// TIA Portal project "AC200_1.1" (V15.1)

(* hardware
DEVICE "S7-1200 station_1"  S7-1200 Station
   slot 0: "Rack_0"  S7-1200 Rack  Rack  V1.0
   slot 1: "PLC_1"  CPU 1215C DC/DC/Rly  6ES7 215-1HG40-0XB0  V4.2
   slot 2: "DI 8x24VDC/DQ 8xRelay_1"  SM 1223 DI8/DQ8 x relay  6ES7 223-1PH32-0XB0  V2.0
   slot 3: "DI 8x24VDC/DQ 8xRelay_2"  SM 1223 DI8/DQ8 x relay  6ES7 223-1PH32-0XB0  V2.0
   slot 4: "AI 4x16BIT_1"  SM 1231 AI4 x HF  6ES7 231-5ND32-0XB0  V2.0
   slot 101: "CM 1241 (RS232)_1"  6ES7 241-1AH32-0XB0  V2.2
DEVICE "HMI_1"  KTP700 Basic PN
   slot 0: "HMI_1"  KTP700 Basic PN  6AV2 123-2GB03-0AX0  15.1.0.0
   slot 1: "HMI_RT_1"  KTP700 Basic PN  6AV2 123-2GB03-0AX0  15.1.0.0
   slot 5: "HMI_1.IE_CP_1"  PROFINET Interface  15.0.1.0
      slot 1: "PROFINET Interface_1"  PROFINET Interface
         slot 1: "Port_1"  Port
*)

// ===== PLC "PLC_1"  CPU 1215C DC/DC/Rly =====

VAR_GLOBAL   // PLC tag table "DI_CPU"
   "DI_EStop_Chain_OK" AT %I0.0 : Bool;   // Nút dừng khẩn NC mắc nối tiếp
   "DI_Phase_OK" AT %I0.1 : Bool;   // Relay bảo vệ mất pha; 1 = nguồn 3 pha tốt
   "DI_Door1_Closed" AT %I0.2 : Bool;   // Công tắc hành trình cửa 1; 1 = cửa đóng
   "DI_Door2_Closed" AT %I0.3 : Bool;   // Công tắc hành trình cửa 2; 1 = cửa đóng
   "DI_Tank_Level_OK" AT %I0.4 : Bool;   // Cảm biến mức bồn nước cấp; 1 = đủ nước
   "DI_SG_Level_High" AT %I0.5 : Bool;   // Mức nước bình sinh hơi; 1 = đầy, 0 = mức thấp
   "DI_GasketPress_High" AT %I0.6 : Bool;   // Tiếp điểm thường mở áp suất cao gioăng cửa; 1 = đạt mức cao
   "DI_JacketPress_High" AT %I0.7 : Bool;   // Tiếp điểm thường mở áp suất cao jacket; 1 = đạt mức cao
   "DI_SGPress_High" AT %I1.0 : Bool;   // Tiếp điểm thường mở áp suất cao bình sinh hơi; 1 = đạt mức cao
   "DI_GasketPress_Low" AT %I1.1 : Bool;
END_VAR

VAR_GLOBAL   // PLC tag table "DI_SM1223_1"
   "DI_Door1_Open_PB" AT %I8.0 : Bool;   // Nút vật lý mở cửa 1
   "DI_Door1_Close_PB" AT %I8.1 : Bool;   // Nút vật lý đóng cửa 1
   "DI_Door2_Open_PB" AT %I8.2 : Bool;   // Nút vật lý mở cửa 2
   "DI_Door2_Close_PB" AT %I8.3 : Bool;   // Nút vật lý đóng cửa 2
   "DI_WaterPump_OL_OK" AT %I8.4 : Bool;   // Tiếp điểm NC relay nhiệt bơm nước; 1 = bình thường
   "DI_VacuumPump_OL_OK" AT %I8.5 : Bool;   // Tiếp điểm NC relay nhiệt bơm chân không; 1 = bình thường
END_VAR

VAR_GLOBAL   // PLC tag table "DO_CPU"
   "DO_Heater1" AT %Q0.0 : Bool;   // Điều khiển SSR cụm nhiệt 9 kW số 1
   "DO_Heater2" AT %Q0.1 : Bool;   // Điều khiển SSR cụm nhiệt 9 kW số 2
   "DO_Heater3" AT %Q0.2 : Bool;   // Điều khiển SSR cụm nhiệt 9 kW số 3
   "DO_WaterPump" AT %Q0.3 : Bool;   // Điều khiển contactor/relay bơm nước
   "DO_VacuumPump" AT %Q0.4 : Bool;   // Điều khiển contactor bơm chân không
   "DO_Door1_Open" AT %Q0.5 : Bool;   // Cuộn mở van 5/2 cửa 1
   "DO_Door1_Close" AT %Q0.6 : Bool;   // Cuộn đóng van 5/2 cửa 1
   "DO_Door2_Open" AT %Q0.7 : Bool;   // Cuộn mở van 5/2 cửa 2
   "DO_Door2_Close" AT %Q1.0 : Bool;   // Cuộn đóng van 5/2 cửa 2
   "DO_Buzzer" AT %Q1.1 : Bool;   // Còi báo 24 VDC
END_VAR

VAR_GLOBAL   // PLC tag table "DO_SM1223_2"
   "DO_WaterInlet_01" AT %Q12.0 : Bool;   // Van điện từ cấp nước NC số 1
   "DO_WaterDrain" AT %Q12.1 : Bool;   // Van điện từ xả nước/khí NO
   "DO_LampRun" AT %Q12.2 : Bool;   // Đèn Run - máy đang vận hành
   "DO_LampError" AT %Q12.3 : Bool;   // Đèn Error - hệ thống có lỗi
   "DO_LampDoor1" AT %Q12.4 : Bool;   // Đèn báo cửa 1 đã đóng an toàn
   "DO_LampDoor2" AT %Q12.5 : Bool;   // Đèn báo cửa 2 đã đóng an toàn
   "DO_WaterInlet_02" AT %Q12.6 : Bool;   // Van điện từ cấp nước NC số 2
END_VAR

VAR_GLOBAL   // PLC tag table "AI_SM1231"
   "AI_ChamberPressure1_Raw" AT %IW128 : Int;   // Áp suất buồng hấp vt1, 4-20 mA, -1...5 bar
   "AI_ChamberPressure2_Raw" AT %IW130 : Int;   // Áp suất buồng hấp vt2, 4-20 mA, -1...5 bar
   "AI_Temperature_Raw" AT %IW132 : Int;   // PT100 qua bộ chuyển đổi 0-10 V
END_VAR

VAR_GLOBAL   // PLC tag table "HMI_Command"
   "HMI_Cmd_Start" AT %M100.0 : Bool;   // Nút Start trên HMI
   "HMI_Cmd_Stop" AT %M100.1 : Bool;   // Dừng bình thường từ HMI
   "HMI_Cmd_Abort" AT %M100.2 : Bool;   // Hủy chu trình từ HMI
   "HMI_Cmd_AckAlarm" AT %M100.3 : Bool;   // Xác nhận cảnh báo và tắt còi
   "HMI_Cmd_Reset" AT %M100.4 : Bool;   // Reset lỗi khi điều kiện đã an toàn
   "HMI_Mode_Auto" AT %M100.5 : Bool;   // Yêu cầu chọn chế độ Auto
   "HMI_Mode_Manual" AT %M100.6 : Bool;   // Yêu cầu chọn chế độ Manual
   "HMI_Mode_Service" AT %M100.7 : Bool;   // Yêu cầu chọn chế độ Service; cần phân quyền
   "HMI_Cmd_Door1Open" AT %M101.0 : Bool;   // Yêu cầu mở cửa 1; PLC phải kiểm tra áp suất và liên động
   "HMI_Cmd_Door1Close" AT %M101.1 : Bool;   // Yêu cầu đóng cửa 1
   "HMI_Cmd_Door2Open" AT %M101.2 : Bool;   // Yêu cầu mở cửa 2; PLC phải kiểm tra áp suất và liên động
   "HMI_Cmd_Door2Close" AT %M101.3 : Bool;   // Yêu cầu đóng cửa 2
   "HMI_Cmd_Print" AT %M101.4 : Bool;   // Yêu cầu in kết quả chu trình
   "HMI_Cmd_ClearAlarmHistory" AT %M101.5 : Bool;   // Yêu cầu xóa lịch sử cảnh báo; cần phân quyền
   "HMI_Cmd_Login" AT %M101.6 : Bool;   // Yêu cầu đăng nhập
   "HMI_Cmd_Logout" AT %M101.7 : Bool;   // Yêu cầu đăng xuất
   "HMI_Cmd_EndAccepted" AT %M121.1 : Bool;
END_VAR

VAR_GLOBAL   // PLC tag table "HMI_Setpoint"
   "HMI_ProgramNumber" AT %MW102 : Int;   // Số chương trình P1-P6
   "HMI_PreVacCycles_SP" AT %MW104 : Int;   // Số lần tiền chân không
   "HMI_SterilizeTime_Min" AT %MW106 : Int;   // Thời gian tiệt trùng, phút
   "HMI_DryTime_Min" AT %MW108 : Int;   // Thời gian sấy, phút
   "HMI_Temperature_SP" AT %MD112 : Real;   // Nhiệt độ đặt, °C
   "HMI_Pressure_SP" AT %MD116 : Real;   // Áp suất đặt, bar
   "HMI_User_Str_Min" AT %MW110 : Int;
   "HMI_User_Dry_Min" AT %MW112 : Int;
   "HMI_User_Temp" AT %MW114 : Int;
END_VAR

VAR_GLOBAL   // PLC tag table "HMI_Status"
   "HMI_Sts_SystemReady" AT %M120.0 : Bool;   // Hệ thống sẵn sàng
   "HMI_Sts_CycleRunning" AT %M120.1 : Bool;   // Chu trình đang chạy
   "HMI_Sts_CycleComplete" AT %M120.2 : Bool;   // Chu trình hoàn thành
   "HMI_Sts_AlarmActive" AT %M120.3 : Bool;   // Đang có cảnh báo
   "HMI_Sts_Door1Closed" AT %M120.4 : Bool;   // Trạng thái cửa 1 đóng
   "HMI_Sts_Door2Closed" AT %M120.5 : Bool;   // Trạng thái cửa 2 đóng
   "HMI_Sts_HeaterRunning" AT %M120.6 : Bool;   // Gia nhiệt đang hoạt động
   "HMI_Sts_VacuumRunning" AT %M120.7 : Bool;   // Bơm chân không đang chạy
   "HMI_ProcessStep" AT %MW122 : Int;   // Mã bước quy trình hiện tại
   "HMI_Temperature_PV" AT %MD124 : Real;   // Nhiệt độ thực tế đã scale, °C
   "HMI_ChamberPressure_01_PV" AT %MD128 : Real;   // Áp suất thực tế buồng hấp tại vị trí 1 đã scale, bar
   "HMI_ChamberPressure_02_PV" AT %MD132 : Real;   // Áp suất thực tế buồng hấp tại vị trí 2 đã scale, bar
   "HMI_RemainingTime_Sec" AT %MD136 : DInt;   // Thời gian còn lại, giây
   "HMI_AlarmErrorWord" AT %MW168 : Int;   // mã loi
   "HMI_ChamberPressure_com" AT %MD144 : Real;   // Ap sau trung binh
   "HMI_Sts_Dry_Enable" AT %M121.0 : Bool;
   "HMI_AlarmWarningWord" AT %MW170 : Int;   // ma canh bao
   "HMI_AlarmAckWord" AT %MW172 : Int;
   "HMI_Sts_BuzzerRequest" AT %M174.0 : Bool;
   "HMI_Sts_LampErrorRequest" AT %M174.1 : Bool;
   "HMI_StartBlockReason" AT %MW174 : Int;
   "HMI_StartBlocked" AT %M174.2 : Bool;
   "HMI_PageRequest" AT %MW176 : Int;
   "HMI_SelectedProgram" AT %MW178 : Int;
END_VAR

VAR_GLOBAL   // PLC tag table "HMI_Manual"
   "HMI_Man_WaterPump" AT %M150.0 : Bool;   // Yêu cầu chạy tay bơm nước; chỉ có hiệu lực trong Service và đủ liên động
   "HMI_Man_VacuumPump" AT %M150.1 : Bool;   // Yêu cầu chạy tay bơm chân không
   "HMI_Man_Heater1" AT %M150.2 : Bool;   // Yêu cầu gia nhiệt tay cụm 1; phải có nước và điều kiện an toàn
   "HMI_Man_Heater2" AT %M150.3 : Bool;   // Yêu cầu gia nhiệt tay cụm 2; phải có nước và điều kiện an toàn
   "HMI_Man_Heater3" AT %M150.4 : Bool;   // Yêu cầu gia nhiệt tay cụm 3; phải có nước và điều kiện an toàn
   "HMI_Man_PilotValve_01" AT %M151.0 : Bool;   // Yêu cầu điều khiển tay van pilot V1; PLC vẫn kiểm tra liên động
   "HMI_Man_PilotValve_02" AT %M151.1 : Bool;   // Yêu cầu điều khiển tay van pilot V2; PLC vẫn kiểm tra liên động
   "HMI_Man_PilotValve_03" AT %M151.2 : Bool;   // Yêu cầu điều khiển tay van pilot V3; PLC vẫn kiểm tra liên động
   "HMI_Man_PilotValve_04" AT %M151.3 : Bool;   // Yêu cầu điều khiển tay van pilot V4; PLC vẫn kiểm tra liên động
   "HMI_Man_PilotValve_05" AT %M151.4 : Bool;   // Yêu cầu điều khiển tay van pilot V5; PLC vẫn kiểm tra liên động
   "HMI_Man_PilotValve_06" AT %M151.5 : Bool;   // Yêu cầu điều khiển tay van pilot V6; PLC vẫn kiểm tra liên động
   "HMI_Man_PilotValve_07" AT %M151.6 : Bool;   // Yêu cầu điều khiển tay van pilot V7; PLC vẫn kiểm tra liên động
   "HMI_Man_PilotValve_08" AT %M151.7 : Bool;   // Yêu cầu điều khiển tay van pilot V8; PLC vẫn kiểm tra liên động
   "HMI_Man_WaterInlet_01" AT %M152.0 : Bool;   // Yêu cầu điều khiển tay van cấp nước 1
   "HMI_Man_WaterDrain" AT %M152.1 : Bool;   // Yêu cầu điều khiển tay van xả
   "HMI_Man_BuzzerTest" AT %M152.2 : Bool;   // Nút thử còi
   "HMI_Man_WaterInlet_02" AT %M152.3 : Bool;   // Yêu cầu chạy thử van cấp nước số 2
END_VAR

VAR_GLOBAL   // PLC tag table "DO_SM1223_1"
   "DO_PilotValve_01" AT %Q8.0 : Bool;   // Van pilot điều khiển van xiên V1
   "DO_PilotValve_02" AT %Q8.1 : Bool;   // Van pilot điều khiển van xiên V2
   "DO_PilotValve_03" AT %Q8.2 : Bool;   // Van pilot điều khiển van xiên V3
   "DO_PilotValve_04" AT %Q8.3 : Bool;   // Van pilot điều khiển van xiên V4/NO
   "DO_PilotValve_05" AT %Q8.4 : Bool;   // Van pilot điều khiển van xiên V5/NO
   "DO_PilotValve_06" AT %Q8.5 : Bool;   // Van pilot điều khiển van xiên V6/NO
   "DO_PilotValve_07" AT %Q8.6 : Bool;   // Van pilot điều khiển van xiên V7/NO
   "DO_PilotValve_08" AT %Q8.7 : Bool;   // Van pilot điều khiển van xiên V8
END_VAR

VAR_GLOBAL   // PLC tag table "Auto_Output"
   "AUTO_Q_Heater1" AT %M164.0 : Bool;   // Đầu ra trung gian Auto cho heater 1; không ghi trực tiếp %Q
   "AUTO_Q_Heater2" AT %M164.1 : Bool;   // Đầu ra trung gian Auto cho heater 2; không ghi trực tiếp %Q
   "AUTO_Q_Heater3" AT %M164.2 : Bool;   // Đầu ra trung gian Auto cho heater 3; không ghi trực tiếp %Q
   "AUTO_Q_WaterPump" AT %M164.3 : Bool;   // Đầu ra trung gian Auto cho bơm nước
   "AUTO_Q_VacuumPump" AT %M164.4 : Bool;   // Đầu ra trung gian Auto cho bơm chân không
   "AUTO_Q_PilotValve_01" AT %M164.5 : Bool;   // Đầu ra trung gian Auto cho van pilot 01
   "AUTO_Q_PilotValve_02" AT %M164.6 : Bool;   // Đầu ra trung gian Auto cho van pilot 02
   "AUTO_Q_PilotValve_03" AT %M164.7 : Bool;   // Đầu ra trung gian Auto cho van pilot 03
   "AUTO_Q_PilotValve_04" AT %M165.0 : Bool;   // Đầu ra trung gian Auto cho van pilot 04
   "AUTO_Q_PilotValve_05" AT %M165.1 : Bool;   // Đầu ra trung gian Auto cho van pilot 05
   "AUTO_Q_PilotValve_06" AT %M165.2 : Bool;   // Đầu ra trung gian Auto cho van pilot 06
   "AUTO_Q_PilotValve_07" AT %M165.3 : Bool;   // Đầu ra trung gian Auto cho van pilot 07
   "AUTO_Q_PilotValve_08" AT %M165.4 : Bool;   // Đầu ra trung gian Auto cho van pilot 08
   "AUTO_Q_WaterInlet_01" AT %M165.5 : Bool;   // Đầu ra trung gian Auto cho van cấp nước 01
   "AUTO_Q_WaterInlet_02" AT %M165.6 : Bool;   // Đầu ra trung gian Auto cho van cấp nước 02
   "AUTO_Q_WaterDrain" AT %M165.7 : Bool;   // Đầu ra trung gian Auto cho van xả nước/khí
   "AUTO_Q_Buzzer" AT %M166.0 : Bool;   // Đầu ra trung gian Auto cho còi báo
   "AUTO_Cmd_Start" AT %M166.1 : Bool;
END_VAR

VAR_GLOBAL   // PLC tag table "Manual_Output"
   "MAN_Q_Heater1" AT %M161.0 : Bool;   // Đầu ra trung gian Manual cho heater 1; không ghi trực tiếp %Q
   "MAN_Q_Heater2" AT %M161.1 : Bool;   // Đầu ra trung gian Manual cho heater 2; không ghi trực tiếp %Q
   "MAN_Q_Heater3" AT %M161.2 : Bool;   // Đầu ra trung gian Manual cho heater 3; không ghi trực tiếp %Q
   "MAN_Q_WaterPump" AT %M161.3 : Bool;   // Đầu ra trung gian Manual cho bơm nước
   "MAN_Q_VacuumPump" AT %M161.4 : Bool;   // Đầu ra trung gian Manual cho bơm chân không
   "MAN_Q_PilotValve_01" AT %M161.5 : Bool;   // Đầu ra trung gian Manual cho van pilot 01
   "MAN_Q_PilotValve_02" AT %M161.6 : Bool;   // Đầu ra trung gian Manual cho van pilot 02
   "MAN_Q_PilotValve_03" AT %M161.7 : Bool;   // Đầu ra trung gian Manual cho van pilot 03
   "MAN_Q_PilotValve_04" AT %M162.0 : Bool;   // Đầu ra trung gian Manual cho van pilot 04
   "MAN_Q_PilotValve_05" AT %M162.1 : Bool;   // Đầu ra trung gian Manual cho van pilot 05
   "MAN_Q_PilotValve_06" AT %M162.2 : Bool;   // Đầu ra trung gian Manual cho van pilot 06
   "MAN_Q_PilotValve_07" AT %M162.3 : Bool;   // Đầu ra trung gian Manual cho van pilot 07
   "MAN_Q_PilotValve_08" AT %M162.4 : Bool;   // Đầu ra trung gian Manual cho van pilot 08
   "MAN_Q_WaterInlet_01" AT %M162.5 : Bool;   // Đầu ra trung gian Manual cho van cấp nước 01
   "MAN_Q_WaterInlet_02" AT %M162.6 : Bool;   // Đầu ra trung gian Manual cho van cấp nước 02
   "MAN_Q_WaterDrain" AT %M162.7 : Bool;   // Đầu ra trung gian Manual cho van xả nước/khí
   "MAN_Q_Buzzer" AT %M163.0 : Bool;   // Đầu ra trung gian Manual cho thử còi
END_VAR

VAR_GLOBAL   // PLC tag table "SIG"
   "SIG_PressureMismatch" AT %M140.0 : Bool;
   "SIG_GasketTimeout" AT %M140.1 : Bool;
   "SIG_Vacuum Timeout" AT %M140.2 : Bool;
   "SIG_Heating Timeout" AT %M140.3 : Bool;
   "SIG_Sterilize TempLow" AT %M140.4 : Bool;
   "SIG_SGFillTimeout" AT %M140.5 : Bool;
   "SIG_ExhaustTimeout" AT %M140.6 : Bool;
   "SIG_Maintenance Due" AT %M140.7 : Bool;
   "SIG_HMICommunicationFault" AT %M141.0 : Bool;
   "SIG_PrinterFault" AT %M141.1 : Bool;
END_VAR

TYPE "UDT_AC200L_AutoConfig"
   STRUCT
      VacuumTarget_bar : Real := -0.75;
      VacuumFallback_bar : Real := -0.65;
      AllowVacuumFallback : Bool := TRUE;
      VacuumTimeout : Time := T#3M;
      ChargeTarget_bar : Real := 0.5;
      ChargeTimeout : Time := T#0MS;   // REQUIRED: not yet specified
      GasketTimeout : Time := T#3M;
      JacketTimeout : Time := T#3M;
      HeatTimeout : Time := T#35M;
      PIDApproach_C : Real := 10.0;
      JacketDrainTime : Time := T#4M;
      SterilizeStableTime : Time := T#0MS;   // REQUIRED
      SterilizePressureMin_bar : Real := 0.0;   // REQUIRED
      SterilizePressureMax_bar : Real := 0.0;   // REQUIRED
      TempLowOffset_C : Real := 1.2;
      TempLowTimeout : Time := T#3M;
      ExhaustTarget_bar : Real := 0.15;
      ExhaustTimeout : Time := T#5M;
      DryTarget_bar : Real := -0.65;
      DryAcquireTimeout : Time := T#0MS;   // REQUIRED
      BalanceTimeout : Time := T#0MS;   // REQUIRED
      ValveSettleTime : Time := T#0MS;   // REQUIRED: mechanical travel time
      PressureSafeBand_bar : Real := 0.15;
      PIDConfigured : Bool := FALSE;   // Set only after PID_Compact configuration
      RecoveryConfigured : Bool := FALSE;   // Confirm recovery exhaust routing
      RunPage : Int := 12;
      EndPage : Int := 15;   // Keep supplied DEMO value, verify actual HMI page
   END_STRUCT;
END_TYPE

DATA_BLOCK "FB_ManualTest_DB"   // DB1
{ S7_Optimized_Access := 'TRUE' }
VERSION : 0.4
// stored: InstanceOfName FB_ManualTest
"FB_ManualTest"
BEGIN
END_DATA_BLOCK

DATA_BLOCK "FB_AC200L_AlarmDirect_V7_DB"   // DB2
{ S7_Optimized_Access := 'TRUE' }
VERSION : 0.1
// stored: InstanceOfName FB_AC200L_AlarmDirect_V7
"FB_AC200L_AlarmDirect_V7"
BEGIN
END_DATA_BLOCK

DATA_BLOCK "FB_AnalogScale_DB"   // DB3
{ S7_Optimized_Access := 'TRUE' }
VERSION : 0.1
// stored: InstanceOfName FB_AnalogScale
"FB_AnalogScale"
BEGIN
END_DATA_BLOCK

DATA_BLOCK "FB_SGStartupFill_DB"   // DB4
{ S7_Optimized_Access := 'TRUE' }
VERSION : 0.5
// stored: InstanceOfName FB_SGStartupFill
"FB_SGStartupFill"
BEGIN
END_DATA_BLOCK

DATA_BLOCK "FB_StartPrecheck_DB"   // DB5
{ S7_Optimized_Access := 'TRUE' }
VERSION : 0.4
// stored: InstanceOfName FB_StartPrecheck
"FB_StartPrecheck"
BEGIN
END_DATA_BLOCK

DATA_BLOCK "FB_AutoCycle_Demo_DB"   // DB6
{ S7_Optimized_Access := 'TRUE' }
VERSION : 0.1
// stored: InstanceOfName FB_AutoCycle_Demo
"FB_AutoCycle_Demo"
BEGIN
END_DATA_BLOCK

DATA_BLOCK "FB_DoorControl_DB"   // DB7
{ S7_Optimized_Access := 'TRUE' }
VERSION : 1.2
// stored: InstanceOfName FB_DoorControl
"FB_DoorControl"
BEGIN
END_DATA_BLOCK

DATA_BLOCK "FB_AutoCycle_Main_DB"   // DB8
{ S7_Optimized_Access := 'TRUE' }
VERSION : 1.3
// stored: InstanceOfName FB_AutoCycle_Main
"FB_AutoCycle_Main"
BEGIN
END_DATA_BLOCK

DATA_BLOCK "DB_AC200L_AutoConfig"   // DB9
{ S7_Optimized_Access := 'TRUE' }
VERSION : 1.0
   VAR
      Settings : "UDT_AC200L_AutoConfig";
   END_VAR
BEGIN
END_DATA_BLOCK

FUNCTION_BLOCK "FB_ManualTest"   // FB1, SCL
{ S7_Optimized_Access := 'TRUE' }
VERSION : 0.4
   VAR_INPUT
      Enable : Bool;
      EStop_OK : Bool;
      Phase_OK : Bool;
      SG_Level_High : Bool;
      WaterPump_OL_OK : Bool;
      VacuumPump_OL_OK : Bool;
      Cmd_Heater1 : Bool;
      Cmd_Heater2 : Bool;
      Cmd_Heater3 : Bool;
      Cmd_WaterPump : Bool;
      Cmd_VacuumPump : Bool;
      Cmd_PilotValve_01 : Bool;
      Cmd_PilotValve_02 : Bool;
      Cmd_PilotValve_03 : Bool;
      Cmd_PilotValve_04 : Bool;
      Cmd_PilotValve_05 : Bool;
      Cmd_PilotValve_06 : Bool;
      Cmd_PilotValve_07 : Bool;
      Cmd_PilotValve_08 : Bool;
      Cmd_WaterInlet_01 : Bool;
      Cmd_WaterInlet_02 : Bool;
      Cmd_WaterDrain : Bool;
      Cmd_Buzzer : Bool;
   END_VAR
   VAR_OUTPUT
      Manual_Ready : Bool;
      Any_Command : Bool;
      Any_Output : Bool;
      Command_Blocked : Bool;
      MoreThanOneCommand : Bool;
      Safety_Trip : Bool;
      Q_Heater1 : Bool;
      Q_Heater2 : Bool;
      Q_Heater3 : Bool;
      Q_WaterPump : Bool;
      Q_VacuumPump : Bool;
      Q_PilotValve_01 : Bool;
      Q_PilotValve_02 : Bool;
      Q_PilotValve_03 : Bool;
      Q_PilotValve_04 : Bool;
      Q_PilotValve_05 : Bool;
      Q_PilotValve_06 : Bool;
      Q_PilotValve_07 : Bool;
      Q_PilotValve_08 : Bool;
      Q_WaterInlet_01 : Bool;
      Q_WaterInlet_02 : Bool;
      Q_WaterDrain : Bool;
      Q_Buzzer : Bool;
   END_VAR
   VAR_TEMP
      CommandCount : Int;
      TestPermit : Bool;
   END_VAR
BEGIN

   #CommandCount := 0;
   IF #Cmd_Heater1 THEN
       #CommandCount := #CommandCount + 1;
   END_IF;
   IF #Cmd_Heater2 THEN
       #CommandCount := #CommandCount + 1;
   END_IF;
   IF #Cmd_Heater3 THEN
       #CommandCount := #CommandCount + 1;
   END_IF;
   IF #Cmd_WaterPump THEN
       #CommandCount := #CommandCount + 1;
   END_IF;
   IF #Cmd_VacuumPump THEN
       #CommandCount := #CommandCount + 1;
   END_IF;
   IF #Cmd_PilotValve_01 THEN
       #CommandCount := #CommandCount + 1;
   END_IF;
   IF #Cmd_PilotValve_02 THEN
       #CommandCount := #CommandCount + 1;
   END_IF;
   IF #Cmd_PilotValve_03 THEN
       #CommandCount := #CommandCount + 1;
   END_IF;
   IF #Cmd_PilotValve_04 THEN
       #CommandCount := #CommandCount + 1;
   END_IF;
   IF #Cmd_PilotValve_05 THEN
       #CommandCount := #CommandCount + 1;
   END_IF;
   IF #Cmd_PilotValve_06 THEN
       #CommandCount := #CommandCount + 1;
   END_IF;
   IF #Cmd_PilotValve_07 THEN
       #CommandCount := #CommandCount + 1;
   END_IF;
   IF #Cmd_PilotValve_08 THEN
       #CommandCount := #CommandCount + 1;
   END_IF;
   IF #Cmd_WaterInlet_01 THEN
       #CommandCount := #CommandCount + 1;
   END_IF;
   IF #Cmd_WaterInlet_02 THEN
       #CommandCount := #CommandCount + 1;
   END_IF;
   IF #Cmd_WaterDrain THEN
       #CommandCount := #CommandCount + 1;
   END_IF;
   IF #Cmd_Buzzer THEN
       #CommandCount := #CommandCount + 1;
   END_IF;
   #Any_Command := #CommandCount > 0;
   #MoreThanOneCommand := #CommandCount > 1;
   #Manual_Ready := #Enable AND #EStop_OK AND #Phase_OK;
   #Safety_Trip := #Enable AND (NOT #EStop_OK OR NOT #Phase_OK);
   #TestPermit := #Manual_Ready;
   #Q_Heater1 := #TestPermit AND #Cmd_Heater1
   AND #SG_Level_High;
   #Q_Heater2 := #TestPermit AND #Cmd_Heater2
   AND #SG_Level_High;
   #Q_Heater3 := #TestPermit AND #Cmd_Heater3
   AND #SG_Level_High;
   #Q_WaterPump := #TestPermit AND #Cmd_WaterPump
   AND #WaterPump_OL_OK;
   #Q_VacuumPump := #TestPermit AND #Cmd_VacuumPump
   AND #VacuumPump_OL_OK;
   #Q_PilotValve_01 := #TestPermit AND #Cmd_PilotValve_01;
   #Q_PilotValve_02 := #TestPermit AND #Cmd_PilotValve_02;
   #Q_PilotValve_03 := #TestPermit AND #Cmd_PilotValve_03;
   #Q_PilotValve_04 := #TestPermit AND #Cmd_PilotValve_04;
   #Q_PilotValve_05 := #TestPermit AND #Cmd_PilotValve_05;
   #Q_PilotValve_06 := #TestPermit AND #Cmd_PilotValve_06;
   #Q_PilotValve_07 := #TestPermit AND #Cmd_PilotValve_07;
   #Q_PilotValve_08 := #TestPermit AND #Cmd_PilotValve_08;
   #Q_WaterInlet_01 := #TestPermit AND #Cmd_WaterInlet_01;
   #Q_WaterInlet_02 := #TestPermit AND #Cmd_WaterInlet_02;
   #Q_WaterDrain := #TestPermit AND #Cmd_WaterDrain;
   #Q_Buzzer := #TestPermit AND #Cmd_Buzzer;
   #Any_Output := #Q_Heater1 OR #Q_Heater2 OR #Q_Heater3
   OR #Q_WaterPump OR #Q_VacuumPump
   OR #Q_PilotValve_01 OR #Q_PilotValve_02
   OR #Q_PilotValve_03 OR #Q_PilotValve_04
   OR #Q_PilotValve_05 OR #Q_PilotValve_06
   OR #Q_PilotValve_07 OR #Q_PilotValve_08
   OR #Q_WaterInlet_01 OR #Q_WaterInlet_02
   OR #Q_WaterDrain OR #Q_Buzzer;
   #Command_Blocked := #Enable AND #Any_Command AND NOT #Any_Output;
END_FUNCTION_BLOCK

FUNCTION_BLOCK "FB_AC200L_AlarmDirect_V7"   // FB2, SCL
{ S7_Optimized_Access := 'TRUE' }
VERSION : 0.1
   VAR_INPUT
      DI_EStop_Chain_OK : Bool;
      DI_Phase_OK : Bool;
      DI_WaterPump_OL_OK : Bool;
      DI_VacuumPump_OL_OK : Bool;
      DI_Tank_Level_OK : Bool;
      DI_Door1_Closed : Bool;
      DI_Door2_Closed : Bool;
      DI_Door1_Open_PB : Bool;
      DI_Door2_Open_PB : Bool;
      AI_Temperature_Raw : Int;
      AI_ChamberPressure1_Raw : Int;
      AI_ChamberPressure2_Raw : Int;
      HMI_Temperature_PV : Real;
      HMI_ChamberPressure_01_PV : Real;
      HMI_ChamberPressure_02_PV : Real;
      HMI_Cmd_Start : Bool;
      HMI_Sts_CycleRunning : Bool;
      SIG_GasketTimeout : Bool;
      SIG_VacuumTimeout : Bool;
      SIG_HeatingTimeout : Bool;
      SIG_SterilizeTempLow : Bool;
      SIG_SGFillTimeout : Bool;
      SIG_ExhaustTimeout : Bool;
      SIG_MaintenanceDue : Bool;
      SIG_HMICommunicationFault : Bool;
      SIG_PrinterFault : Bool;
      SIG_PressureMismatch : Bool;
   END_VAR
   VAR_OUTPUT
      AlarmErrorWord : Int;
      AlarmWarningWord : Int;
      ErrorActive : Bool;
      WarningActive : Bool;
      AlarmActive : Bool;
      LampErrorRequest : Bool;
      BuzzerRequest : Bool;
   END_VAR
   VAR_IN_OUT
      AlarmAckWord : Int;
   END_VAR
   VAR
      TankLowTimer : TON_TIME;
   END_VAR
   VAR_TEMP
      UnackError : Bool;
   END_VAR
BEGIN
       #AlarmErrorWord.%X0 := NOT #DI_EStop_Chain_OK;
       #AlarmErrorWord.%X1 := NOT #DI_Phase_OK;
       #AlarmErrorWord.%X2 := NOT #DI_WaterPump_OL_OK;
       #AlarmErrorWord.%X3 := NOT #DI_VacuumPump_OL_OK;
       #AlarmErrorWord.%X4 := #HMI_Temperature_PV > 138.0;

       #TankLowTimer(
                     IN := NOT #DI_Tank_Level_OK,
                     PT := T#15s
       );

       #AlarmErrorWord.%X5 := #TankLowTimer.Q;

       #AlarmErrorWord.%X6 := (#AI_Temperature_Raw < 0)
       OR (#AI_Temperature_Raw > 27648);

       #AlarmErrorWord.%X7 := (#AI_ChamberPressure1_Raw < 0)
       OR (#AI_ChamberPressure1_Raw > 27648);

       #AlarmErrorWord.%X8 := (#AI_ChamberPressure2_Raw < 0)
       OR (#AI_ChamberPressure2_Raw > 27648);

       #AlarmErrorWord.%X9 := #SIG_PressureMismatch;
       #AlarmErrorWord.%X10 := #SIG_GasketTimeout;
       #AlarmErrorWord.%X11 := #SIG_VacuumTimeout;
       #AlarmErrorWord.%X12 := #SIG_HeatingTimeout;
       #AlarmErrorWord.%X13 := #SIG_SterilizeTempLow;
       #AlarmErrorWord.%X14 := #SIG_SGFillTimeout;
       #AlarmErrorWord.%X15 := #SIG_ExhaustTimeout;

       #AlarmWarningWord.%X0 := #HMI_Sts_CycleRunning
       AND #DI_Door1_Open_PB;

       #AlarmWarningWord.%X1 := #HMI_Sts_CycleRunning
       AND #DI_Door2_Open_PB;

       #AlarmWarningWord.%X2 := #HMI_Cmd_Start
       AND ((NOT #DI_Door1_Closed)
       OR (NOT #DI_Door2_Closed));

       #AlarmWarningWord.%X3 := (#DI_Door1_Open_PB OR #DI_Door2_Open_PB)
       AND ((#HMI_ChamberPressure_01_PV < -0.15)
       OR (#HMI_ChamberPressure_01_PV > 0.15)
       OR (#HMI_ChamberPressure_02_PV < -0.15)
       OR (#HMI_ChamberPressure_02_PV > 0.15));

       #AlarmWarningWord.%X4 := #SIG_MaintenanceDue;
       #AlarmWarningWord.%X5 := #SIG_HMICommunicationFault;
       #AlarmWarningWord.%X6 := #SIG_PrinterFault;
       #AlarmWarningWord.%X7 := FALSE;
       #AlarmWarningWord.%X8 := FALSE;
       #AlarmWarningWord.%X9 := FALSE;
       #AlarmWarningWord.%X10 := FALSE;
       #AlarmWarningWord.%X11 := FALSE;
       #AlarmWarningWord.%X12 := FALSE;
       #AlarmWarningWord.%X13 := FALSE;
       #AlarmWarningWord.%X14 := FALSE;
       #AlarmWarningWord.%X15 := FALSE;

       #ErrorActive := #AlarmErrorWord.%X0
       OR #AlarmErrorWord.%X1
       OR #AlarmErrorWord.%X2
       OR #AlarmErrorWord.%X3
       OR #AlarmErrorWord.%X4
       OR #AlarmErrorWord.%X5
       OR #AlarmErrorWord.%X6
       OR #AlarmErrorWord.%X7
       OR #AlarmErrorWord.%X8
       OR #AlarmErrorWord.%X9
       OR #AlarmErrorWord.%X10
       OR #AlarmErrorWord.%X11
       OR #AlarmErrorWord.%X12
       OR #AlarmErrorWord.%X13
       OR #AlarmErrorWord.%X14
       OR #AlarmErrorWord.%X15;

       #WarningActive := #AlarmWarningWord.%X0
       OR #AlarmWarningWord.%X1
       OR #AlarmWarningWord.%X2
       OR #AlarmWarningWord.%X3
       OR #AlarmWarningWord.%X4
       OR #AlarmWarningWord.%X5
       OR #AlarmWarningWord.%X6;

       #AlarmActive := #ErrorActive OR #WarningActive;

       #AlarmAckWord.%X0 := #AlarmAckWord.%X0 AND #AlarmErrorWord.%X0;
       #AlarmAckWord.%X1 := #AlarmAckWord.%X1 AND #AlarmErrorWord.%X1;
       #AlarmAckWord.%X2 := #AlarmAckWord.%X2 AND #AlarmErrorWord.%X2;
       #AlarmAckWord.%X3 := #AlarmAckWord.%X3 AND #AlarmErrorWord.%X3;
       #AlarmAckWord.%X4 := #AlarmAckWord.%X4 AND #AlarmErrorWord.%X4;
       #AlarmAckWord.%X5 := #AlarmAckWord.%X5 AND #AlarmErrorWord.%X5;
       #AlarmAckWord.%X6 := #AlarmAckWord.%X6 AND #AlarmErrorWord.%X6;
       #AlarmAckWord.%X7 := #AlarmAckWord.%X7 AND #AlarmErrorWord.%X7;
       #AlarmAckWord.%X8 := #AlarmAckWord.%X8 AND #AlarmErrorWord.%X8;
       #AlarmAckWord.%X9 := #AlarmAckWord.%X9 AND #AlarmErrorWord.%X9;
       #AlarmAckWord.%X10 := #AlarmAckWord.%X10 AND #AlarmErrorWord.%X10;
       #AlarmAckWord.%X11 := #AlarmAckWord.%X11 AND #AlarmErrorWord.%X11;
       #AlarmAckWord.%X12 := #AlarmAckWord.%X12 AND #AlarmErrorWord.%X12;
       #AlarmAckWord.%X13 := #AlarmAckWord.%X13 AND #AlarmErrorWord.%X13;
       #AlarmAckWord.%X14 := #AlarmAckWord.%X14 AND #AlarmErrorWord.%X14;
       #AlarmAckWord.%X15 := #AlarmAckWord.%X15 AND #AlarmErrorWord.%X15;

       #UnackError :=
       (#AlarmErrorWord.%X0 AND NOT #AlarmAckWord.%X0)
       OR (#AlarmErrorWord.%X1 AND NOT #AlarmAckWord.%X1)
       OR (#AlarmErrorWord.%X2 AND NOT #AlarmAckWord.%X2)
       OR (#AlarmErrorWord.%X3 AND NOT #AlarmAckWord.%X3)
       OR (#AlarmErrorWord.%X4 AND NOT #AlarmAckWord.%X4)
       OR (#AlarmErrorWord.%X5 AND NOT #AlarmAckWord.%X5)
       OR (#AlarmErrorWord.%X6 AND NOT #AlarmAckWord.%X6)
       OR (#AlarmErrorWord.%X7 AND NOT #AlarmAckWord.%X7)
       OR (#AlarmErrorWord.%X8 AND NOT #AlarmAckWord.%X8)
       OR (#AlarmErrorWord.%X9 AND NOT #AlarmAckWord.%X9)
       OR (#AlarmErrorWord.%X10 AND NOT #AlarmAckWord.%X10)
       OR (#AlarmErrorWord.%X11 AND NOT #AlarmAckWord.%X11)
       OR (#AlarmErrorWord.%X12 AND NOT #AlarmAckWord.%X12)
       OR (#AlarmErrorWord.%X13 AND NOT #AlarmAckWord.%X13)
       OR (#AlarmErrorWord.%X14 AND NOT #AlarmAckWord.%X14)
       OR (#AlarmErrorWord.%X15 AND NOT #AlarmAckWord.%X15);

       #LampErrorRequest := #ErrorActive;
       #BuzzerRequest := #UnackError <> 0;
END_FUNCTION_BLOCK

FUNCTION_BLOCK "FB_AnalogScale"   // FB3, SCL
{ S7_Optimized_Access := 'TRUE' }
VERSION : 0.1
   VAR_INPUT
      Pressure01_Raw : Int;
      Pressure02_Raw : Int;
      Temperature_Raw : Int;
      TempAt0V_C : Real;
      TempAt10V_C : Real;
   END_VAR
   VAR_OUTPUT
      Pressure01_bar : Real;
      Pressure02_bar : Real;
      PressureAvg_bar : Real;
      Temperature_C : Real;
      PressureMismatchFault : Bool;
      PressuresAgree : Bool;
      BothNearZero : Bool;
   END_VAR
   VAR
      DiffTimer : TON_TIME;
   END_VAR
   VAR_TEMP
      Mismatch : Bool;
   END_VAR
BEGIN
       // Scale two 4-20 mA pressure transmitters, -1 to +5 bar.
       #Pressure01_bar := -1.0 + INT_TO_REAL(#Pressure01_Raw) * 6.0 / 27648.0;
       #Pressure02_bar := -1.0 + INT_TO_REAL(#Pressure02_Raw) * 6.0 / 27648.0;
       #PressureAvg_bar := (#Pressure01_bar + #Pressure02_bar) / 2.0;

       // PT100 transmitter: 0 V = TempAt0V_C; 10 V = TempAt10V_C.
       #Temperature_C := #TempAt0V_C + INT_TO_REAL(#Temperature_Raw)
       * (#TempAt10V_C - #TempAt0V_C) / 27648.0;

       // The existing alarm block checks raw sensor faults separately.
       #Mismatch := ABS(#Pressure01_bar - #Pressure02_bar) > 0.3;
       #DiffTimer(IN := #Mismatch,
                  PT := T#10s);
       #PressureMismatchFault := #DiffTimer.Q;
       #PressuresAgree := NOT #Mismatch;

       // This is only a pressure condition; also require no sensor faults
       // and the remaining door interlocks in the output control block.
       #BothNearZero := #PressuresAgree
       AND (#Pressure01_bar > -0.1) AND (#Pressure01_bar < 0.1)
       AND (#Pressure02_bar > -0.1) AND (#Pressure02_bar < 0.1);
END_FUNCTION_BLOCK

FUNCTION_BLOCK "FB_SGStartupFill"   // FB4, SCL
{ S7_Optimized_Access := 'TRUE' }
VERSION : 0.5
   VAR_INPUT
      Enable : Bool;
      ManualTestActive : Bool;
      SGLevelHigh : Bool;
      SGPressHigh : Bool;
      TankLevelOK : Bool;
      WaterPumpOLOK : Bool;
      EStopChainOK : Bool;
      PhaseOK : Bool;
   END_VAR
   VAR_OUTPUT
      FillRequest : Bool;
      HeatRequest : Bool;
      SteamReady : Bool;
      FillTimeoutFault : Bool;
      FillElapsed : Time;
      HeatRequest3 : Bool;
   END_VAR
   VAR
      FillTimer : TON_TIME;
      FirstHeatDone : Bool;
   END_VAR
   VAR_TEMP
      RunAuto : Bool;
   END_VAR
BEGIN
       #RunAuto := #Enable AND NOT #ManualTestActive;

       // The 5-minute window starts when the controller enables filling
       // with the steam generator below its high-level probe.
       // An empty supply tank does not pause this window.
       #FillTimer(IN := #RunAuto AND NOT #SGLevelHigh AND NOT #FillTimeoutFault,
                  PT := T#5m,
                  ET => #FillElapsed);

       IF #FillTimer.Q THEN
           #FillTimeoutFault := TRUE;
       END_IF;

       // Clear the timeout only after the generator reaches the high level.
       // Manual Test can be used to fill it after a timeout.
       IF #SGLevelHigh THEN
           #FillTimeoutFault := FALSE;
       END_IF;

       #FillRequest := #RunAuto
       AND #EStopChainOK
       AND #PhaseOK
       AND #TankLevelOK
       AND #WaterPumpOLOK
       AND NOT #SGLevelHigh
       AND NOT #FillTimeoutFault;

       // Preheat ends when the high steam pressure switch first operates.
       // A later pressure drop must not automatically restart startup heating.
       IF NOT #RunAuto AND NOT #SGPressHigh THEN
           #SteamReady := FALSE;
       ELSIF #SGPressHigh AND #SGLevelHigh THEN
           #SteamReady := TRUE;
       END_IF;

       // If the high-level probe drops, heating stops and filling resumes.
       IF #RunAuto AND #SGLevelHigh AND #SGPressHigh THEN
           #FirstHeatDone := TRUE;
       END_IF;

       #HeatRequest := #RunAuto
       AND #EStopChainOK
       AND #PhaseOK
       AND #TankLevelOK
       AND #SGLevelHigh
       AND NOT #SGPressHigh
       AND NOT #FillTimeoutFault;

       #HeatRequest3 := #HeatRequest AND NOT #FirstHeatDone;
END_FUNCTION_BLOCK

FUNCTION_BLOCK "FB_StartPrecheck"   // FB5, SCL
{ S7_Optimized_Access := 'TRUE' }
VERSION : 0.4
   VAR_INPUT
      AutoMode : Bool;
      Door1Closed : Bool;
      Door2Closed : Bool;
      PhaseOK : Bool;
      EStopChainOK : Bool;
      SGLevelHigh : Bool;
      SGPressHigh : Bool;
      TankLevelOK : Bool;
      ManualTestActive : Bool;
      CycleRunning : Bool;
      ErrorActive : Bool;
   END_VAR
   VAR_OUTPUT
      ReadyToStart : Bool;
      StartAccepted : Bool;
      StartBlocked : Bool;
      BlockReason : Int;
   END_VAR
   VAR_IN_OUT
      HMI_Cmd_Start : Bool;
   END_VAR
BEGIN
       // All green indicators must be TRUE before a cycle can start.
       #ReadyToStart := #AutoMode
       AND NOT #ManualTestActive
       AND #EStopChainOK AND #PhaseOK
       AND #Door1Closed AND #Door2Closed
       AND #TankLevelOK AND #SGLevelHigh AND #SGPressHigh
       AND NOT #CycleRunning AND NOT #ErrorActive;

       // Output a one-scan pulse to the auto cycle only after a valid press.
       #StartAccepted := FALSE;

       // HMI sets HMI_Cmd_Start ONCE on press; PLC clears it after reading.
       IF #HMI_Cmd_Start THEN
           #HMI_Cmd_Start := FALSE;

           IF #ReadyToStart THEN
               #StartAccepted := TRUE;
               #StartBlocked := FALSE;
               #BlockReason := 0;
           ELSE
               #StartBlocked := TRUE;

               IF NOT #AutoMode OR #ManualTestActive THEN
                   #BlockReason := 9; // Auto mode unavailable / Manual Test active
               ELSIF NOT #EStopChainOK THEN
                   #BlockReason := 1;
               ELSIF NOT #PhaseOK THEN
                   #BlockReason := 2;
               ELSIF NOT #Door1Closed THEN
                   #BlockReason := 3;
               ELSIF NOT #Door2Closed THEN
                   #BlockReason := 4;
               ELSIF NOT #TankLevelOK THEN
                   #BlockReason := 5;
               ELSIF NOT #SGLevelHigh THEN
                   #BlockReason := 6;
               ELSIF NOT #SGPressHigh THEN
                   #BlockReason := 7;
               ELSIF #CycleRunning THEN
                   #BlockReason := 12;
               ELSIF #ErrorActive THEN
                   #BlockReason := 10;
               END_IF;
           END_IF;
       END_IF;
END_FUNCTION_BLOCK

FUNCTION_BLOCK "FB_AutoCycle_Demo"   // FB6, SCL
{ S7_Optimized_Access := 'TRUE' }
VERSION : 0.1
// AC200L: timed HMI/PLC cycle demo only. No process actuator is commanded.
//  Call once per OB1 scan, AFTER FB_StartPrecheck and BEFORE FC_OutputControl.
//  OB1 connections (symbol names from the supplied PLC tag tables):
//    StartAccepted     := "AUTO_Cmd_Start" (FB_StartPrecheck.StartAccepted)
//    AbortCmd          := "HMI_Cmd_Abort"       [InOut]
//    ProgramNumber     := "HMI_ProgramNumber"
//    CycleRunning      => "HMI_Sts_CycleRunning"
//    CycleComplete     => "HMI_Sts_CycleComplete"
//    ProcessStep       => "HMI_ProcessStep"
//    RemainingTimeMin  => "HMI_RemainingTime_Sec" (existing DInt tag)
//    PageRequest       := "HMI_PageRequest"     [InOut]
//    BuzzerRequest     => "AUTO_Q_Buzzer"
//  HMI_RemainingTime_Sec is a legacy name. It now carries whole MINUTES
//  (ceil of the remaining seconds) for the washing-machine style display.
//  Do NOT enable HMI scaling; show zero decimal places and label the field min.
//  For clarity, rename this PLC/HMI tag to HMI_RemainingTime_Min later if desired.
//  Shared End screen: ResultCode, CompletedProgram, StartTime, EndTime.
//  ResultCode: 0=none, 1=complete, 2=cancelled by operator.
//  StartTime and EndTime are DTL snapshots of the PLC local clock.
//  Show dates only when TimeStampsValid is TRUE.
//  Text_list_step mapping: 0=Idle, 1=Vacuum, 2=Heating,
//  3=Sterilization, 4=Exhaust, 5=Drying.
//  Keep FB_SGStartupFill in the current project. This FB does not touch its
//  existing FillRequest and HeatRequest outputs. Use PLCSIM for the cycle demo.
//  Keep the original alarm FB unchanged: it alone writes HMI_Sts_BuzzerRequest.
//  Existing FC_OutputControl ORs HMI_Sts_BuzzerRequest with AUTO_Q_Buzzer.
   VAR_INPUT
      StartAccepted : Bool;
      ProgramNumber : Int;
      ErrorActive : Bool;
   END_VAR
   VAR_OUTPUT
      CycleRunning : Bool;
      CycleComplete : Bool;
      ResultCode : Int;
      ProcessStep : Int;
      RemainingTimeMin : DInt;
      CompletedProgram : Int;
      CompletedTimeSec : DInt;
      StartTime : DTL;
      EndTime : DTL;
      TimeStampsValid : Bool;
      BuzzerRequest : Bool;
   END_VAR
   VAR_IN_OUT
      AbortCmd : Bool;
      PageRequest : Int;
   END_VAR
   VAR
      Phase1Timer : TON_TIME;
      Phase2Timer : TON_TIME;
      Phase3Timer : TON_TIME;
      Phase4Timer : TON_TIME;
      Phase5Timer : TON_TIME;
      TotalTimer : TON_TIME;
      FinishTimer : TON_TIME;
      BeepActive : Bool;
      ActiveProgram : Int;
      StartClockValid : Bool;
   END_VAR
   VAR_TEMP
      Phase1Enable : Bool;
      Phase2Enable : Bool;
      Phase3Enable : Bool;
      Phase4Enable : Bool;
      Phase5Enable : Bool;
      Phase1Done : Bool;
      Phase2Done : Bool;
      Phase3Done : Bool;
      Phase4Done : Bool;
      Phase5Done : Bool;
      FinishDone : Bool;
      Phase1Elapsed : Time;
      Phase2Elapsed : Time;
      Phase3Elapsed : Time;
      Phase4Elapsed : Time;
      Phase5Elapsed : Time;
      TotalElapsed : Time;
      BeepElapsed : Time;
      RemainingMs : DInt;
      ClockNow : DTL;
      ClockStatus : Int;
   END_VAR
BEGIN
       // Call all timer instances on every scan. Inactive phases reset.
       #Phase1Enable := #CycleRunning AND (#ProcessStep = 1);
       #Phase2Enable := #CycleRunning AND (#ProcessStep = 2);
       #Phase3Enable := #CycleRunning AND (#ProcessStep = 3);
       #Phase4Enable := #CycleRunning AND (#ProcessStep = 4);
       #Phase5Enable := #CycleRunning AND (#ProcessStep = 5);

       #Phase1Timer(IN := #Phase1Enable,
                    PT := T#5s,
                    Q => #Phase1Done,
                    ET => #Phase1Elapsed);
       #Phase2Timer(IN := #Phase2Enable,
                    PT := T#5s,
                    Q => #Phase2Done,
                    ET => #Phase2Elapsed);
       #Phase3Timer(IN := #Phase3Enable,
                    PT := T#5s,
                    Q => #Phase3Done,
                    ET => #Phase3Elapsed);
       #Phase4Timer(IN := #Phase4Enable,
                    PT := T#5s,
                    Q => #Phase4Done,
                    ET => #Phase4Elapsed);
       #Phase5Timer(IN := #Phase5Enable,
                    PT := T#5s,
                    Q => #Phase5Done,
                    ET => #Phase5Elapsed);
       #TotalTimer(IN := #CycleRunning,
                   PT := T#1h,
                   ET => #TotalElapsed);
       #FinishTimer(IN := #BeepActive,
                    PT := T#5s,
                    Q => #FinishDone,
                    ET => #BeepElapsed);

       IF #ErrorActive AND #CycleRunning THEN
           #AbortCmd := FALSE;
           #CompletedProgram := #ActiveProgram;
           #CompletedTimeSec := TIME_TO_DINT(#TotalElapsed) / 1000;

           #TimeStampsValid := FALSE;
           #ClockStatus := RD_LOC_T(OUT => #ClockNow);

           IF ((#ClockStatus = 0) OR (#ClockStatus = 1))
               AND #StartClockValid THEN
               #EndTime := #ClockNow;
               #TimeStampsValid := TRUE;
           END_IF;

           #CycleRunning := FALSE;
           #CycleComplete := FALSE;
           #ResultCode := 3;       // Stopped due to error
           #ProcessStep := 0;
           #BeepActive := FALSE;    // Alarm block control buzzer
           #ActiveProgram := 0;
           #PageRequest := 15;     // End screen

       // Abort takes priority. The precheck block alone consumes HMI_Cmd_Start;
       // this block consumes only the confirmed HMI_Cmd_Abort command.
       ELSIF #AbortCmd THEN
           #AbortCmd := FALSE;
           IF #CycleRunning THEN
               // Save the interrupted cycle before resetting its running state.
               #CompletedProgram := #ActiveProgram;
               #CompletedTimeSec := TIME_TO_DINT(#TotalElapsed) / 1000;
               #TimeStampsValid := FALSE;
               #ClockStatus := RD_LOC_T(OUT => #ClockNow);
               IF ((#ClockStatus = 0) OR (#ClockStatus = 1)) AND #StartClockValid THEN
                   #EndTime := #ClockNow;
                   #TimeStampsValid := TRUE;
               END_IF;
               #CycleRunning := FALSE;
               #CycleComplete := FALSE;
               #ResultCode := 2;
               #ProcessStep := 0;
               #BeepActive := FALSE;
               #ActiveProgram := 0;
               #PageRequest := 15;
           END_IF;

       ELSIF #StartAccepted AND NOT #CycleRunning THEN
           #CycleRunning := TRUE;
           #CycleComplete := FALSE;
           #ResultCode := 0;
           #ProcessStep := 1;
           #CompletedProgram := 0;
           #CompletedTimeSec := 0;
           #StartClockValid := FALSE;
           #TimeStampsValid := FALSE;
           #BeepActive := FALSE;
           #ActiveProgram := #ProgramNumber;
           #ClockStatus := RD_LOC_T(OUT => #ClockNow);
           IF (#ClockStatus = 0) OR (#ClockStatus = 1) THEN
               #StartTime := #ClockNow;
               #StartClockValid := TRUE;
           END_IF;
           #PageRequest := 12;   // Existing running screen

       ELSIF #CycleRunning THEN
           CASE #ProcessStep OF
               1:  // Vacuum (display only)
                   IF #Phase1Done THEN
                       #ProcessStep := 2;
                   END_IF;
               2:  // Heating (display only)
                   IF #Phase2Done THEN
                       #ProcessStep := 3;
                   END_IF;
               3:  // Sterilization (display only)
                   IF #Phase3Done THEN
                       #ProcessStep := 4;
                   END_IF;
               4:  // Exhaust (display only)
                   IF #Phase4Done THEN
                       #ProcessStep := 5;
                   END_IF;
               5:  // Drying (display only)
                   IF #Phase5Done THEN
                       #CompletedProgram := #ActiveProgram;
                       #CompletedTimeSec := TIME_TO_DINT(#TotalElapsed) / 1000;
                       #ClockStatus := RD_LOC_T(OUT => #ClockNow);
                       IF ((#ClockStatus = 0) OR (#ClockStatus = 1)) AND #StartClockValid THEN
                           #EndTime := #ClockNow;
                           #TimeStampsValid := TRUE;
                       END_IF;
                       #CycleRunning := FALSE;
                       #CycleComplete := TRUE;
                       #ResultCode := 1;
                       #ProcessStep := 0;
                       #BeepActive := TRUE;
                       #PageRequest := 15;  // Configure completion screen as ID 15
                   END_IF;
               ELSE
                   // An unexpected step is treated as an abort, never completion.
                   #CycleRunning := FALSE;
                   #CycleComplete := FALSE;
                   #ResultCode := 0;
                   #ProcessStep := 0;
                   #BeepActive := FALSE;
                   #TimeStampsValid := FALSE;
                   #PageRequest := 15;
           END_CASE;
       END_IF;

       // Calculate the remaining time of the CURRENT step after the state
       // transition, so the display immediately shows 1 min for the new step.
       #RemainingMs := 0;
       IF #CycleRunning THEN
           CASE #ProcessStep OF
               1:
                   #RemainingMs := 5000 - TIME_TO_DINT(#Phase1Elapsed);
               2:
                   #RemainingMs := 5000 - TIME_TO_DINT(#Phase2Elapsed);
               3:
                   #RemainingMs := 5000 - TIME_TO_DINT(#Phase3Elapsed);
               4:
                   #RemainingMs := 5000 - TIME_TO_DINT(#Phase4Elapsed);
               5:
                   #RemainingMs := 5000 - TIME_TO_DINT(#Phase5Elapsed);
           END_CASE;
       END_IF;
       IF #RemainingMs < 0 THEN
           #RemainingMs := 0;
       END_IF;
       // 1..60000 ms = 1 min; 60001..120000 ms = 2 min; zero = 0 min.
       #RemainingTimeMin := (#RemainingMs + 59999) / 60000;

       // ON: [0,1), [2,3), [4,5) s. OFF: [1,2), [3,4) s and after 5 s.
       IF #FinishDone THEN
           #BeepActive := FALSE;
       END_IF;
       #BuzzerRequest := #BeepActive AND NOT #AbortCmd AND
       ((#BeepElapsed < T#1s) OR
       ((#BeepElapsed >= T#2s) AND (#BeepElapsed < T#3s)) OR
       ((#BeepElapsed >= T#4s) AND (#BeepElapsed < T#5s)));
END_FUNCTION_BLOCK

FUNCTION_BLOCK "FB_DoorControl"   // FB7, SCL
{ S7_Optimized_Access := 'TRUE' }
VERSION : 1.2
// AC200L - two-door hold-to-run control. Call every scan before FC_OutputControl.
//  This FB does not own the alarm word, alarm acknowledgement or event history.
   VAR_INPUT
      EStopOK : Bool;
      PhaseOK : Bool;
      CycleActive : Bool;   // TRUE from accepted Start through preparation/end
      Door1Closed : Bool;
      Door2Closed : Bool;
      GasketPressHigh : Bool;
      Pressure1_bar : Real;
      Pressure2_bar : Real;
      Door1OpenPB : Bool;
      Door1ClosePB : Bool;
      Door2OpenPB : Bool;
      Door2ClosePB : Bool;
   END_VAR
   VAR_OUTPUT
      Door1OpenCmd : Bool;
      Door1CloseCmd : Bool;
      Door2OpenCmd : Bool;
      Door2CloseCmd : Bool;
      Door1OpenBlocked : Bool;   // Level TRUE while blocked Open1 PB is held
      Door2OpenBlocked : Bool;   // Level TRUE while blocked Open2 PB is held
      DoorCommandBlocked : Bool;   // Any actionable door command rejected
      DoorFaultDuringRun : Bool;   // Door-closed feedback lost during cycle
   END_VAR
   VAR_TEMP
      PressureSafe : Bool;
      Conflict : Bool;
      Close1Blocked : Bool;
      Close2Blocked : Bool;
   END_VAR
BEGIN
       // Sensor diagnostics are handled by the separate alarm block.
       // Both measured chamber pressures must be near atmospheric pressure.
       #PressureSafe := (#Pressure1_bar >= -0.15)
       AND (#Pressure1_bar <= 0.15)
       AND (#Pressure2_bar >= -0.15)
       AND (#Pressure2_bar <= 0.15);

       // Deny contradictory directions and simultaneous movement of both doors.
       #Conflict := (#Door1OpenPB AND #Door1ClosePB)
       OR (#Door2OpenPB AND #Door2ClosePB)
       OR ((#Door1OpenPB OR #Door1ClosePB)
       AND (#Door2OpenPB OR #Door2ClosePB));

       #Door1OpenCmd := #EStopOK AND #PhaseOK AND NOT #CycleActive
       AND NOT #Conflict AND #Door1OpenPB
       AND #Door2Closed AND NOT #GasketPressHigh
       AND #PressureSafe;
       #Door2OpenCmd := #EStopOK AND #PhaseOK AND NOT #CycleActive
       AND NOT #Conflict AND #Door2OpenPB
       AND #Door1Closed AND NOT #GasketPressHigh
       AND #PressureSafe;

       // A door may be closed even when the other door is still open.
       #Door1CloseCmd := #EStopOK AND #PhaseOK AND NOT #CycleActive
       AND NOT #Conflict AND #Door1ClosePB AND NOT #Door1Closed;
       #Door2CloseCmd := #EStopOK AND #PhaseOK AND NOT #CycleActive
       AND NOT #Conflict AND #Door2ClosePB AND NOT #Door2Closed;

       // These are status signals. FB_AlarmDirect decides whether/how to warn,
       // latch, acknowledge and log them; this FB never writes HMI_AlarmWord.
       #Door1OpenBlocked := #Door1OpenPB AND NOT #Door1OpenCmd;
       #Door2OpenBlocked := #Door2OpenPB AND NOT #Door2OpenCmd;
       #Close1Blocked := #Door1ClosePB AND NOT #Door1CloseCmd AND NOT #Door1Closed;
       #Close2Blocked := #Door2ClosePB AND NOT #Door2CloseCmd AND NOT #Door2Closed;
       #DoorCommandBlocked := #Door1OpenBlocked OR #Door2OpenBlocked
       OR #Close1Blocked OR #Close2Blocked;
       #DoorFaultDuringRun := #CycleActive
       AND (NOT #Door1Closed OR NOT #Door2Closed);
END_FUNCTION_BLOCK

FUNCTION_BLOCK "FB_AutoCycle_Main"   // FB8, SCL
{ S7_Optimized_Access := 'TRUE' }
VERSION : 1.3
// AC200L process sequence, OB1 once per scan. All Q_Valve requests mean OPEN.
//  Only FC_OutputControl writes hardware DO. PID_Compact runs in cyclic OB.
//  CTAS10 = jacket pressure switch; gauge16 has NO electrical feedback.
   VAR_INPUT
      StartAccepted : Bool;
      AutoMode : Bool;
      EStopOK : Bool;
      PhaseOK : Bool;
      ErrorActive : Bool;   // Process-stopping errors only, not warnings
      Door1Closed : Bool;
      Door2Closed : Bool;
      GasketPressHigh : Bool;
      JacketPressHigh : Bool;   // CTAS10, NEVER chamber pressure
      AlarmErrorWord : Int;   // Read existing Alarm diagnostics, bits X6..X9
      Temperature_C : Real;
      Pressure1_bar : Real;
      Pressure2_bar : Real;
      ProgramNumber : Int;   // 1..5 preset, 6 User
      SP_Temp_C : Real;
      SP_Sterilize_min : Int;
      SP_DryEnable : Bool;
      SP_Dry_min : Int;
      PumpPermit : Bool;   // overload + inlet pressure/temperature limits
      Door1OpenPB : Bool;   // DI_Door1_Open_PB
      Door2OpenPB : Bool;   // DI_Door2_Open_PB
      GasketReleasedConfirmed : Bool;   // proven depressurized; NOT NOT CTAS12
      PIDPulse : Bool;   // PID_Compact.Output_PWM, never connect directly to DO
      PIDError : DWord;
      Config : "UDT_AC200L_AutoConfig";
   END_VAR
   VAR_OUTPUT
      CycleRunning : Bool;
      CycleActive : Bool;   // door/mode lock through recovery and safe finish
      CycleComplete : Bool;
      ProcessStep : Int;   // 0 prep/idle,1 vacuum,2 heat,3 hold,4 exhaust,5 dry,6 balance
      SubStep : Int;
      ResultCode : Int;   // 0 none,1 complete,2 cancel,3 fault
      FaultCode : Int;
      ConfigValid : Bool;
      StartRejected : Bool;
      EndAcceptBlocked : Bool;
      CompletedProgram : Int;
      CompletedTimeSec : DInt;
      RemainingTimeMin : DInt;
      RemainingIsTimeout : Bool;
      SterilizeElapsedSec : DInt;
      DryElapsedSec : DInt;
      TempMin_C : Real;
      TempMax_C : Real;
      TempExtremaValid : Bool;
      TempLowActive : Bool;
      VacuumFallbackUsed : Bool;
      VacuumPulsesDone : Int;
      ActiveTemp_C : Real;
      ActiveSterilize_min : Int;
      ActiveDry_min : Int;
      StartTime : DTL;
      EndTime : DTL;
      TimeStampsValid : Bool;
      PIDEnable : Bool;
      BuzzerRequest : Bool;
      StopSGHeating : Bool;
      DoorReleasePermitted : Bool;
      Q_VacuumPump : Bool;
      Q_PilotValve_01 : Bool;   // jacket steam
      Q_PilotValve_02 : Bool;   // gasket supply
      Q_PilotValve_03 : Bool;   // chamber steam, PID
      Q_PilotValve_04 : Bool;   // HEPA
      Q_PilotValve_05 : Bool;   // SG drain, no automatic opening
      Q_PilotValve_06 : Bool;   // chamber vacuum/exhaust
      Q_PilotValve_07 : Bool;   // jacket drain
      Q_PilotValve_08 : Bool;   // gasket drain NC
      Q_WaterInlet_01 : Bool;   // HX cooling water
      Q_WaterDrain : Bool;
   END_VAR
   VAR_IN_OUT
      AbortCmd : Bool;
      PageRequest : Int;
      EndAccepted : Bool;   // End-screen close/return command, NOT alarm Ack
   END_VAR
   VAR
      Cfg : "UDT_AC200L_AutoConfig";
      TotalTimer : TON_TIME;
      StageTimer : TON_TIME;
      GasketTimer : TON_TIME;
      JacketTimer : TON_TIME;
      JacketDrainTimer : TON_TIME;
      StableTimer : TON_TIME;
      TempLowTimer : TON_TIME;
      DryAcquireTimer : TON_TIME;
      BalanceTimer : TON_TIME;
      RecoveryIsolationTimer : TON_TIME;
      FinishTimer : TON_TIME;
      PreviousStep : Int;
      PreviousTotalMs : DInt;
      HoldMs : DInt;
      DryMs : DInt;
      PulsesRequired : Int;
      PIDSwitched : Bool;
      SealHeld : Bool;
      SealReleasing : Bool;
      BeepActive : Bool;
      StartClockValid : Bool;
      PreviousHoldQualified : Bool;
      PreviousDryQualified : Bool;
   END_VAR
   VAR_TEMP
      SensorsOK : Bool;   // derived from Alarm; NO raw checks in Auto
      CommonOK : Bool;
      PressureOK : Bool;
      PressureSafe : Bool;
      HoldQualified : Bool;
      DryQualified : Bool;
      HeatStable : Bool;
      JacketDemand : Bool;
      ChangedStep : Bool;
      StagePT : Time;
      TotalMs : DInt;
      DeltaMs : DInt;
      RemainingMs : DInt;
      EventResult : Int;
      NewFault : Int;
      ClockStatus : Int;
      ClockNow : DTL;
   END_VAR
BEGIN
   // Alarm is the sole owner of raw sensor diagnostics.
   // Use its specific bits so an unrelated cycle timeout does not prevent recovery.
   #SensorsOK := NOT #AlarmErrorWord.%X6 AND NOT #AlarmErrorWord.%X7
   AND NOT #AlarmErrorWord.%X8 AND NOT #AlarmErrorWord.%X9;
   #CommonOK := #EStopOK AND #PhaseOK;
   #PressureOK := #SensorsOK AND (ABS(#Pressure1_bar - #Pressure2_bar) <= 0.3);
   #ConfigValid := (#Config.GasketTimeout > T#0ms)
   AND (#Config.JacketTimeout > T#0ms) AND (#Config.ChargeTimeout > T#0ms)
   AND (#Config.VacuumTimeout > T#0ms) AND (#Config.HeatTimeout > T#0ms)
   AND (#Config.SterilizeStableTime > T#0ms)
   AND (#Config.ExhaustTimeout > T#0ms) AND (#Config.BalanceTimeout > T#0ms)
   AND (#Config.DryAcquireTimeout > T#0ms) AND (#Config.ValveSettleTime > T#0ms)
   AND (#Config.JacketDrainTime > T#0ms) AND (#Config.TempLowTimeout > T#0ms)
   AND (#Config.VacuumTarget_bar >= -1.0)
   AND (#Config.VacuumTarget_bar < #Config.VacuumFallback_bar)
   AND (#Config.VacuumFallback_bar < 0.0)
   AND (#Config.ChargeTarget_bar > 0.0)
   AND (#Config.DryTarget_bar >= -1.0) AND (#Config.DryTarget_bar < 0.0)
   AND (#Config.PressureSafeBand_bar > 0.0) AND (#Config.PressureSafeBand_bar <= 0.15)
   AND (#Config.ExhaustTarget_bar > 0.0) AND (#Config.ExhaustTarget_bar <= 0.15)
   AND (#Config.SterilizePressureMin_bar > 0.0)
   AND (#Config.SterilizePressureMax_bar > #Config.SterilizePressureMin_bar)
   AND (#Config.PIDApproach_C > 0.0) AND (#Config.TempLowOffset_C > 0.0)
   AND #Config.PIDConfigured AND #Config.RecoveryConfigured;
   #PressureSafe := #PressureOK
   AND (ABS(#Pressure1_bar) <= 0.15) AND (ABS(#Pressure2_bar) <= 0.15);
   #StartRejected := FALSE;
   #EndAcceptBlocked := FALSE;
   #EventResult := 0;
   #NewFault := 0;

   // Elapsed-ms delta is derived from a Siemens monotonic timer, not wall clock.
   #TotalTimer(IN := #CycleActive,
               PT := T#24d);
   #TotalMs := TIME_TO_DINT(#TotalTimer.ET);
   #DeltaMs := #TotalMs - #PreviousTotalMs;
   IF #DeltaMs < 0 THEN
       #DeltaMs := 0;
   END_IF;
   #PreviousTotalMs := #TotalMs;

   #ChangedStep := #SubStep <> #PreviousStep;
   #PreviousStep := #SubStep;
   #StagePT := T#24d;
   CASE #SubStep OF
       11:
           #StagePT := #Cfg.VacuumTimeout;
       12, 14, 42, 60:
           #StagePT := #Cfg.ValveSettleTime;
       13:
           #StagePT := #Cfg.ChargeTimeout;
       20:
           #StagePT := #Cfg.HeatTimeout;
       40:
           #StagePT := #Cfg.ExhaustTimeout;
   END_CASE;
   #StageTimer(IN := #CycleRunning AND NOT #ChangedStep,
               PT := #StagePT);

   #JacketDemand := #CycleRunning
   AND (((#SubStep = 20) AND NOT #PIDSwitched)
   OR ((#SubStep = 50) OR (#SubStep = 51)))
   AND NOT (#PIDSwitched AND NOT #JacketDrainTimer.Q);
   #GasketTimer(IN := #CycleRunning AND #SealHeld AND NOT #GasketPressHigh,
                PT := #Cfg.GasketTimeout);
   #JacketTimer(IN := #JacketDemand AND NOT #JacketPressHigh,
                PT := #Cfg.JacketTimeout);
   // Latched event, independent of HMI step. Continues across heating/hold/exhaust.
   #JacketDrainTimer(IN := #CycleActive AND #PIDSwitched AND (#ResultCode = 0),
                     PT := #Cfg.JacketDrainTime);
   #HeatStable := #CycleRunning AND (#SubStep = 20) AND #PressureOK
   AND #GasketPressHigh AND (#Temperature_C >= #ActiveTemp_C)
   AND (#Pressure1_bar >= #Cfg.SterilizePressureMin_bar)
   AND (#Pressure2_bar >= #Cfg.SterilizePressureMin_bar)
   AND (#Pressure1_bar <= #Cfg.SterilizePressureMax_bar)
   AND (#Pressure2_bar <= #Cfg.SterilizePressureMax_bar)
   AND (#PIDError = DWORD#0);
   #StableTimer(IN := #HeatStable,
                PT := #Cfg.SterilizeStableTime);
   #TempLowActive := #CycleRunning AND (#SubStep = 30)
   AND (#Temperature_C < (#ActiveTemp_C - #Cfg.TempLowOffset_C));
   #TempLowTimer(IN := #TempLowActive,
                 PT := #Cfg.TempLowTimeout);
   #HoldQualified := #CycleRunning AND (#SubStep = 30) AND #PressureOK
   AND #GasketPressHigh AND NOT #TempLowActive AND (#PIDError = DWORD#0)
   AND (#Pressure1_bar >= #Cfg.SterilizePressureMin_bar)
   AND (#Pressure2_bar >= #Cfg.SterilizePressureMin_bar)
   AND (#Pressure1_bar <= #Cfg.SterilizePressureMax_bar)
   AND (#Pressure2_bar <= #Cfg.SterilizePressureMax_bar);
   #DryQualified := #CycleRunning AND (#SubStep = 51) AND #PressureOK
   AND #PumpPermit AND #GasketPressHigh
   AND (#Pressure1_bar <= #Cfg.DryTarget_bar)
   AND (#Pressure2_bar <= #Cfg.DryTarget_bar);
   #DryAcquireTimer(IN := #CycleRunning AND ((#SubStep = 50) OR (#SubStep = 51))
                    AND NOT (#PressureOK AND (#Pressure1_bar <= #Cfg.DryTarget_bar)
                    AND (#Pressure2_bar <= #Cfg.DryTarget_bar)),
                    PT := #Cfg.DryAcquireTimeout);
   #BalanceTimer(IN := #CycleActive AND ((#SubStep = 61) OR (#SubStep = 90)),
                 PT := #Cfg.BalanceTimeout);
   #RecoveryIsolationTimer(IN := #CycleActive AND (#SubStep = 90),
                           PT := #Cfg.ValveSettleTime);
   #FinishTimer(IN := #BeepActive,
                PT := T#5s);

   // Reset cycle timeout memory only after the end has been safely accepted.
   // External errors remain authoritative. This command is not alarm Ack.
   IF #EndAccepted THEN
       #EndAccepted := FALSE;
       IF NOT #CycleActive AND (#ResultCode <> 0) AND #PressureSafe
           AND #CommonOK THEN
           #FaultCode := 0;
           #StopSGHeating := FALSE;
       ELSE
           #EndAcceptBlocked := TRUE;
       END_IF;
   END_IF;

   IF #CycleRunning THEN
       IF #TempExtremaValid AND (#SubStep = 30) AND #SensorsOK THEN
           IF #Temperature_C < #TempMin_C THEN
               #TempMin_C := #Temperature_C;
           END_IF;
           IF #Temperature_C > #TempMax_C THEN
               #TempMax_C := #Temperature_C;
           END_IF;
       END_IF;
       IF #HoldQualified AND #PreviousHoldQualified THEN
           #HoldMs := #HoldMs + #DeltaMs;
       END_IF;
       IF #DryQualified AND #PreviousDryQualified THEN
           #DryMs := #DryMs + #DeltaMs;
       END_IF;
       IF #ErrorActive OR NOT #CommonOK OR NOT #SensorsOK THEN
           #NewFault := 1;
       ELSIF NOT #AutoMode THEN
           #NewFault := 2;
       ELSIF ((#SubStep = 11) OR (#SubStep = 50) OR (#SubStep = 51))
           AND NOT #PumpPermit THEN
           #NewFault := 5;
       ELSIF NOT #Door1Closed OR NOT #Door2Closed THEN
           #NewFault := 3;
       ELSIF #GasketTimer.Q THEN
           #NewFault := 10;
       ELSIF #JacketTimer.Q THEN
           #NewFault := 11;
       ELSIF #PIDSwitched AND (#PIDError <> DWORD#0) THEN
           #NewFault := 12;
       ELSIF #TempLowTimer.Q THEN
           #NewFault := 13;
       ELSIF #DryAcquireTimer.Q THEN
           #NewFault := 14;
       ELSIF #TotalTimer.Q THEN
           #NewFault := 15;
       END_IF;
   END_IF;
   IF #NewFault <> 0 THEN
       #EventResult := 3;
   ELSIF #AbortCmd AND #CycleRunning THEN
       #EventResult := 2;
   END_IF;

   IF (#EventResult = 0) AND #CycleRunning AND #GasketPressHigh THEN
       CASE #SubStep OF
           10: // initial seal; no pump before CTAS12
               IF #GasketPressHigh THEN
                   #SubStep := 11;
               END_IF;
           11: // vacuum pulse; evaluate CURRENT values of BOTH sensors
               IF #PressureOK AND (#Pressure1_bar <= #Cfg.VacuumTarget_bar)
                   AND (#Pressure2_bar <= #Cfg.VacuumTarget_bar) THEN
                   #SubStep := 12;
               ELSIF #StageTimer.Q THEN
                   IF #Cfg.AllowVacuumFallback AND #PressureOK
                       AND (#Pressure1_bar <= #Cfg.VacuumFallback_bar)
                       AND (#Pressure2_bar <= #Cfg.VacuumFallback_bar) THEN
                       #VacuumFallbackUsed := TRUE;
                       #SubStep := 12;
                   ELSE
                       #NewFault := 20;
                   END_IF;
               END_IF;
           12:
               IF #StageTimer.Q THEN
                   #SubStep := 13;
               END_IF; // isolate suction
           13: // charge steam, count only completed vacuum+charge pairs
               IF #PressureOK AND (#Pressure1_bar >= #Cfg.ChargeTarget_bar)
                   AND (#Pressure2_bar >= #Cfg.ChargeTarget_bar) THEN
                   #VacuumPulsesDone := #VacuumPulsesDone + 1;
                   IF #VacuumPulsesDone >= #PulsesRequired THEN
                       #SubStep := 20;
                   ELSE
                       #SubStep := 14;
                   END_IF;
               ELSIF #StageTimer.Q THEN
                   #NewFault := 21;
               END_IF;
           14:
               IF #StageTimer.Q THEN
                   #SubStep := 11;
               END_IF; // close steam before suction
           20:
               IF #Temperature_C >= (#ActiveTemp_C - #Cfg.PIDApproach_C) THEN
                   #PIDSwitched := TRUE;
               END_IF;
               IF #StableTimer.Q THEN
                   #SubStep := 30;
                   #HoldMs := 0;
                   #TempMin_C := #Temperature_C;
                   #TempMax_C := #Temperature_C;
                   #TempExtremaValid := TRUE;
               ELSIF #StageTimer.Q THEN
                   #NewFault := 22;
               END_IF;
           30:
               IF #PressureOK AND ((#Pressure1_bar < #Cfg.SterilizePressureMin_bar)
                   OR (#Pressure2_bar < #Cfg.SterilizePressureMin_bar)
                   OR (#Pressure1_bar > #Cfg.SterilizePressureMax_bar)
                   OR (#Pressure2_bar > #Cfg.SterilizePressureMax_bar)) THEN
                   #NewFault := 23;
               ELSIF #HoldMs >= (INT_TO_DINT(#ActiveSterilize_min) * 60000) THEN
                   #SubStep := 42;
               END_IF;
           42:
               IF #StageTimer.Q THEN
                   #SubStep := 40;
               END_IF;
           40:
               IF #PressureOK AND (#Pressure1_bar < #Cfg.ExhaustTarget_bar)
                   AND (#Pressure2_bar < #Cfg.ExhaustTarget_bar) THEN
                   IF #ActiveDry_min > 0 THEN
                       // Never feed jacket while its drain task is still active.
                       IF #JacketDrainTimer.Q THEN
                           #SubStep := 50;
                       END_IF;
                   ELSE
                       #SubStep := 60;
                   END_IF;
               ELSIF #StageTimer.Q THEN
                   #NewFault := 24;
               END_IF;
           50:
               IF #PressureOK AND #PumpPermit
                   AND (#Pressure1_bar <= #Cfg.DryTarget_bar)
                   AND (#Pressure2_bar <= #Cfg.DryTarget_bar) THEN
                   #SubStep := 51;
               END_IF;
           51:
               IF #DryMs >= (INT_TO_DINT(#ActiveDry_min) * 60000) THEN
                   #SubStep := 60;
               END_IF;
           60:
               IF #StageTimer.Q THEN
                   #SubStep := 61;
               END_IF;
           61:
               IF #PressureOK AND (ABS(#Pressure1_bar) <= #Cfg.PressureSafeBand_bar)
                   AND (ABS(#Pressure2_bar) <= #Cfg.PressureSafeBand_bar)
               THEN
                   #EventResult := 1;
               ELSIF #BalanceTimer.Q THEN
                   #NewFault := 25;
               END_IF;
           ELSE
               #NewFault := 99;
       END_CASE;
   END_IF;
   IF #NewFault <> 0 THEN
       #EventResult := 3;
   END_IF;

   IF #EventResult <> 0 THEN
       #ResultCode := #EventResult;
       #FaultCode := #NewFault;
       #CycleRunning := FALSE;
       #CycleComplete := #EventResult = 1;
       #CompletedTimeSec := #TotalMs / 1000;
       #TimeStampsValid := FALSE;
       #ClockStatus := RD_LOC_T(OUT => #ClockNow);
       IF ((#ClockStatus = 0) OR (#ClockStatus = 1)) AND #StartClockValid THEN
           #EndTime := #ClockNow;
           #TimeStampsValid := TRUE;
       END_IF;
       #PageRequest := #Cfg.EndPage;
       #BeepActive := #EventResult = 1;
       IF #EventResult = 1 THEN
           #CycleActive := FALSE;
           #SubStep := 0;
       ELSE
           #StopSGHeating := TRUE;
           #SubStep := 90; // retain lock through pressure recovery
       END_IF;
   END_IF;

   IF #CycleActive AND (#SubStep = 90) THEN
       IF #PressureSafe AND #CommonOK THEN
           #CycleActive := FALSE;
           #SubStep := 0;
       END_IF;
       // Recovery timeout never releases door or marks the cycle complete.
       IF #BalanceTimer.Q AND (#FaultCode = 0) THEN
           #FaultCode := 26;
       END_IF;
   END_IF;

   IF #StartAccepted AND NOT #CycleActive AND (#EventResult = 0) AND NOT #AbortCmd THEN
       IF #ConfigValid AND #AutoMode AND #CommonOK AND NOT #ErrorActive
           AND #PressureSafe AND #Door1Closed AND #Door2Closed
           AND (#FaultCode = 0) AND NOT #SealReleasing
           AND (#ProgramNumber >= 1) AND (#ProgramNumber <= 6)
           AND (#SP_Temp_C >= 110.0) AND (#SP_Temp_C <= 134.0)
           AND (#SP_Sterilize_min >= 1) AND (#SP_Sterilize_min <= 99)
           AND (#SP_Dry_min >= 0) AND (#SP_Dry_min <= 99) THEN
           #Cfg := #Config; // freeze process configuration for the entire run
           #ActiveTemp_C := #SP_Temp_C;
           #ActiveSterilize_min := #SP_Sterilize_min;
           #ActiveDry_min := 0;
           IF #SP_DryEnable THEN
               #ActiveDry_min := #SP_Dry_min;
           END_IF;
           #CompletedProgram := #ProgramNumber;
           #PulsesRequired := 4;
           IF (#ProgramNumber = 1) OR (#ProgramNumber = 2) OR (#ProgramNumber = 5) THEN
               #PulsesRequired := 3;
           END_IF;
           #CycleRunning := TRUE;
           #CycleActive := TRUE;
           #CycleComplete := FALSE;
           #ResultCode := 0;
           #SubStep := 10;
           #SealHeld := TRUE;
           #PIDSwitched := FALSE;
           #VacuumFallbackUsed := FALSE;
           #VacuumPulsesDone := 0;
           #HoldMs := 0;
           #DryMs := 0;
           #PreviousTotalMs := 0;
           #PreviousHoldQualified := FALSE;
           #PreviousDryQualified := FALSE;
           #TempExtremaValid := FALSE;
           #TempMin_C := 0.0;
           #TempMax_C := 0.0;
           #CompletedTimeSec := 0;
           #TimeStampsValid := FALSE;
           #BeepActive := FALSE;
           #ClockStatus := RD_LOC_T(OUT => #ClockNow);
           #StartClockValid := (#ClockStatus = 0) OR (#ClockStatus = 1);
           IF #StartClockValid THEN
               #StartTime := #ClockNow;
           END_IF;
           #PageRequest := #Cfg.RunPage;
       ELSE
           #StartRejected := TRUE;
       END_IF;
   END_IF;
   #AbortCmd := FALSE;
   #PreviousHoldQualified := #HoldQualified AND (#SubStep = 30) AND #CycleRunning;
   #PreviousDryQualified := #DryQualified AND (#SubStep = 51) AND #CycleRunning;

   // Deterministic defaults. Electrical NO inversion belongs ONLY to OutputControl.
   #Q_VacuumPump := FALSE;
   #Q_PilotValve_01 := FALSE;
   #Q_PilotValve_02 := FALSE;
   #Q_PilotValve_03 := FALSE;
   #Q_PilotValve_04 := FALSE;
   #Q_PilotValve_05 := FALSE;
   #Q_PilotValve_06 := FALSE;
   #Q_PilotValve_07 := FALSE;
   #Q_PilotValve_08 := FALSE;
   #Q_WaterInlet_01 := FALSE;
   #Q_WaterDrain := FALSE;
   #PIDEnable := #CycleRunning AND #PIDSwitched AND #CommonOK AND #AutoMode
   AND NOT #ErrorActive AND #SensorsOK AND ((#SubStep = 20) OR (#SubStep = 30));
   IF #CycleRunning AND #CommonOK AND #AutoMode AND NOT #ErrorActive AND #SensorsOK THEN
       // Pause process actuation if seal pressure is not proven; recovery timeout still runs.
       #Q_PilotValve_02 := #SealHeld AND NOT #GasketPressHigh;
       IF #GasketPressHigh THEN
           CASE #SubStep OF
               11, 50, 51:
                   #Q_PilotValve_06 := TRUE;
                   #Q_VacuumPump := #PumpPermit;
                   #Q_WaterInlet_01 := TRUE;
                   #Q_WaterDrain := TRUE;
               13:
                   #Q_PilotValve_03 := TRUE;
               20:
                   #Q_PilotValve_03 := NOT #PIDSwitched OR (#PIDPulse AND (#PIDError = DWORD#0));
                   #Q_PilotValve_01 := NOT #PIDSwitched AND NOT #JacketPressHigh;
               30:
                   #Q_PilotValve_03 := #PIDPulse AND (#PIDError = DWORD#0);
               40:
                   #Q_PilotValve_06 := TRUE;
                   #Q_WaterInlet_01 := TRUE;
                   #Q_WaterDrain := TRUE;
               61:
                   IF #PressureOK THEN
                       IF (#Pressure1_bar > #Cfg.PressureSafeBand_bar)
                           OR (#Pressure2_bar > #Cfg.PressureSafeBand_bar) THEN
                           #Q_PilotValve_06 := TRUE;
                           #Q_WaterInlet_01 := TRUE;
                           #Q_WaterDrain := TRUE;
                       ELSIF (#Pressure1_bar < - #Cfg.PressureSafeBand_bar)
                           OR (#Pressure2_bar < - #Cfg.PressureSafeBand_bar) THEN
                           #Q_PilotValve_04 := TRUE;
                       END_IF;
                   END_IF;
           END_CASE;
           IF #PIDSwitched AND NOT #JacketDrainTimer.Q AND (#SubStep <> 60) AND (#SubStep <> 61) THEN
               #Q_PilotValve_07 := TRUE;
               #Q_WaterInlet_01 := TRUE;
               #Q_WaterDrain := TRUE;
           END_IF;
           IF ((#SubStep = 50) OR (#SubStep = 51)) AND #JacketDrainTimer.Q THEN
               #Q_PilotValve_01 := NOT #JacketPressHigh;
           END_IF;
       END_IF;
   END_IF;
   IF (#SubStep = 90) AND #CycleActive AND #CommonOK AND #PressureOK
       AND #Cfg.RecoveryConfigured
       AND #RecoveryIsolationTimer.Q THEN
       IF (#Pressure1_bar > #Cfg.PressureSafeBand_bar)
           OR (#Pressure2_bar > #Cfg.PressureSafeBand_bar) THEN
           #Q_PilotValve_06 := TRUE;
           #Q_WaterInlet_01 := TRUE;
           #Q_WaterDrain := TRUE;
       ELSIF (#Pressure1_bar < - #Cfg.PressureSafeBand_bar)
           OR (#Pressure2_bar < - #Cfg.PressureSafeBand_bar) THEN
           #Q_PilotValve_04 := TRUE;
       END_IF;
   END_IF;

   // Do not release the seal at cycle-end automatically. Explicit OPEN request only.
   IF NOT #CycleActive AND (#Door1OpenPB OR #Door2OpenPB) AND #PressureSafe
       AND #CommonOK AND NOT #GasketReleasedConfirmed THEN
       #SealReleasing := TRUE;
       #SealHeld := FALSE;
   END_IF;
   IF #SealReleasing AND #CommonOK AND #PressureSafe THEN
       #Q_PilotValve_08 := NOT #GasketReleasedConfirmed;
       IF #GasketReleasedConfirmed THEN
           #SealReleasing := FALSE;
       END_IF;
   END_IF;
   #DoorReleasePermitted := NOT #CycleActive AND #PressureSafe
   AND #GasketReleasedConfirmed AND #CommonOK;
   // Maintain seal after COMPLETED until operator explicitly requests opening.
   IF #SealHeld AND NOT #CycleActive AND (#ResultCode = 1) AND #CommonOK THEN
       #Q_PilotValve_02 := NOT #GasketPressHigh;
   END_IF;

   #ProcessStep := 0;
   CASE #SubStep OF
       11, 12, 13, 14:
           #ProcessStep := 1;
       20:
           #ProcessStep := 2;
       30:
           #ProcessStep := 3;
       40, 42:
           #ProcessStep := 4;
       50, 51:
           #ProcessStep := 5;
       60, 61, 90:
           #ProcessStep := 6;
   END_CASE;
   #RemainingMs := 0;
   #RemainingIsTimeout := TRUE;
   #StagePT := T#24d;
   CASE #SubStep OF
       11:
           #StagePT := #Cfg.VacuumTimeout;
       12, 14, 42, 60:
           #StagePT := #Cfg.ValveSettleTime;
       13:
           #StagePT := #Cfg.ChargeTimeout;
       20:
           #StagePT := #Cfg.HeatTimeout;
       40:
           #StagePT := #Cfg.ExhaustTimeout;
   END_CASE;
   IF #CycleRunning THEN
       CASE #SubStep OF
           10:
               #RemainingMs := TIME_TO_DINT(#Cfg.GasketTimeout - #GasketTimer.ET);
           11, 12, 13, 14, 20, 40, 42, 60:
               #RemainingMs := TIME_TO_DINT(#StagePT - #StageTimer.ET);
           30:
               #RemainingMs := INT_TO_DINT(#ActiveSterilize_min) * 60000 - #HoldMs;
               #RemainingIsTimeout := FALSE;
           50:
               #RemainingMs := TIME_TO_DINT(#Cfg.DryAcquireTimeout - #DryAcquireTimer.ET);
           51:
               #RemainingMs := INT_TO_DINT(#ActiveDry_min) * 60000 - #DryMs;
               #RemainingIsTimeout := FALSE;
           61:
               #RemainingMs := TIME_TO_DINT(#Cfg.BalanceTimeout - #BalanceTimer.ET);
       END_CASE;
   END_IF;
   IF #CycleRunning AND (#SubStep <> #PreviousStep) THEN
       CASE #SubStep OF
           11, 12, 13, 14, 20, 40, 42, 60:
               #RemainingMs := TIME_TO_DINT(#StagePT);
           50:
               #RemainingMs := TIME_TO_DINT(#Cfg.DryAcquireTimeout);
           61:
               #RemainingMs := TIME_TO_DINT(#Cfg.BalanceTimeout);
       END_CASE;
   END_IF;
   IF #RemainingMs < 0 THEN
       #RemainingMs := 0;
   END_IF;
   #RemainingTimeMin := #RemainingMs / 60000;
   IF (#RemainingMs MOD 60000) > 0 THEN
       #RemainingTimeMin := #RemainingTimeMin + 1;
   END_IF;
   #SterilizeElapsedSec := #HoldMs / 1000;
   #DryElapsedSec := #DryMs / 1000;
   IF #FinishTimer.Q THEN
       #BeepActive := FALSE;
   END_IF;
   #BuzzerRequest := #BeepActive AND NOT #ErrorActive
   AND ((#FinishTimer.ET < T#1s)
   OR ((#FinishTimer.ET >= T#2s) AND (#FinishTimer.ET < T#3s))
   OR ((#FinishTimer.ET >= T#4s) AND (#FinishTimer.ET < T#5s)));
END_FUNCTION_BLOCK

FUNCTION "FC_OutputControl" : Void   // FC1, SCL
{ S7_Optimized_Access := 'TRUE' }
VERSION : 0.5
   VAR_TEMP
      Common_OK : Bool;
      Heater_OK : Bool;
      DoorPressureSafe : Bool;
      AnyManualOutput : Bool;
      AnyAutoOutput : Bool;
      ManualMode : Bool;
      AutoMode : Bool;
   END_VAR
BEGIN
   // DO_PilotValve_04,05,06,07 and DO_WaterDrain control NO valves

   #ManualMode := "HMI_Mode_Manual" AND NOT "HMI_Mode_Auto";
   #AutoMode := "HMI_Mode_Auto" AND NOT "HMI_Mode_Manual";

   #Common_OK := "DI_EStop_Chain_OK" AND "DI_Phase_OK";
   #Heater_OK := #Common_OK
   AND "DI_Tank_Level_OK"
   AND "DI_SG_Level_High"
   AND NOT "DI_SGPress_High"
   AND NOT "SIG_SGFillTimeout";

   #DoorPressureSafe := ("HMI_ChamberPressure_com" >= -0.10)
   AND ("HMI_ChamberPressure_com" <= 0.10);

   "DO_Heater1" := #Heater_OK
   AND ((#ManualMode AND "MAN_Q_Heater1")
   OR (#AutoMode AND "AUTO_Q_Heater1")
   OR (NOT "HMI_Mode_Manual" AND "FB_SGStartupFill_DB".HeatRequest));
   "DO_Heater2" := #Heater_OK
   AND ((#ManualMode AND "MAN_Q_Heater2")
   OR (#AutoMode AND "AUTO_Q_Heater2")
   OR (NOT "HMI_Mode_Manual" AND "FB_SGStartupFill_DB".HeatRequest ));
   "DO_Heater3" := #Heater_OK
   AND ((#ManualMode AND "MAN_Q_Heater3")
   OR (#AutoMode AND "AUTO_Q_Heater3")
   OR (NOT "HMI_Mode_Manual" AND "FB_SGStartupFill_DB".HeatRequest3));

   "DO_WaterPump" := #Common_OK
   AND "DI_Tank_Level_OK"
   AND "DI_WaterPump_OL_OK"
   AND (("FB_SGStartupFill_DB".FillRequest)
   OR (#ManualMode AND "MAN_Q_WaterPump")
   OR (#AutoMode AND "AUTO_Q_WaterPump"));
   "DO_VacuumPump" := #Common_OK
   AND "DI_VacuumPump_OL_OK"
   AND ((#ManualMode AND "MAN_Q_VacuumPump")
   OR (#AutoMode AND "AUTO_Q_VacuumPump"));

   "DO_PilotValve_01" := #Common_OK
   AND ((#ManualMode AND "MAN_Q_PilotValve_01")
   OR (#AutoMode AND "AUTO_Q_PilotValve_01"));
   "DO_PilotValve_02" := #Common_OK
   AND ((#ManualMode AND "MAN_Q_PilotValve_02")
   OR (#AutoMode AND "AUTO_Q_PilotValve_02"));
   "DO_PilotValve_03" := #Common_OK
   AND ((#ManualMode AND "MAN_Q_PilotValve_03")
   OR (#AutoMode AND "AUTO_Q_PilotValve_03"));

   "DO_PilotValve_04" := #Common_OK
   AND NOT ((#ManualMode AND "MAN_Q_PilotValve_04")
   OR (#AutoMode AND "AUTO_Q_PilotValve_04"));
   "DO_PilotValve_05" := #Common_OK
   AND NOT ((#ManualMode AND "MAN_Q_PilotValve_05")
   OR (#AutoMode AND "AUTO_Q_PilotValve_05"));
   "DO_PilotValve_06" := #Common_OK
   AND NOT ((#ManualMode AND "MAN_Q_PilotValve_06")
   OR (#AutoMode AND "AUTO_Q_PilotValve_06"));
   "DO_PilotValve_07" := #Common_OK
   AND NOT ((#ManualMode AND "MAN_Q_PilotValve_07")
   OR (#AutoMode AND "AUTO_Q_PilotValve_07"));

   "DO_PilotValve_08" := #Common_OK
   AND ((#ManualMode AND "MAN_Q_PilotValve_08")
   OR (#AutoMode AND "AUTO_Q_PilotValve_08"));

   "DO_WaterInlet_01" := #Common_OK
   AND ((#ManualMode AND "MAN_Q_WaterInlet_01")
   OR (#AutoMode AND "AUTO_Q_WaterInlet_01"));
   "DO_WaterInlet_02" := #Common_OK
   AND ((#ManualMode AND "MAN_Q_WaterInlet_02")
   OR (#AutoMode AND "AUTO_Q_WaterInlet_02")
   OR (NOT "HMI_Mode_Manual" AND "FB_SGStartupFill_DB".FillRequest));
   "DO_WaterDrain" := #Common_OK
   AND NOT ((#ManualMode AND "MAN_Q_WaterDrain")
   OR (#AutoMode AND "AUTO_Q_WaterDrain"));

   "DO_Door1_Open" := "FB_DoorControl_DB".Door1OpenCmd;
   "DO_Door1_Close" := "FB_DoorControl_DB".Door1CloseCmd;
   "DO_Door2_Open" := "FB_DoorControl_DB".Door2OpenCmd;
   "DO_Door2_Close" := "FB_DoorControl_DB".Door2CloseCmd;

   "DO_Buzzer" :="HMI_Sts_BuzzerRequest"
   OR (#ManualMode AND "MAN_Q_Buzzer")
   OR (#AutoMode AND "AUTO_Q_Buzzer");

   #AnyManualOutput := "MAN_Q_Heater1" OR "MAN_Q_Heater2" OR "MAN_Q_Heater3"
   OR "MAN_Q_WaterPump" OR "MAN_Q_VacuumPump"
   OR "MAN_Q_PilotValve_01" OR "MAN_Q_PilotValve_02"
   OR "MAN_Q_PilotValve_03" OR "MAN_Q_PilotValve_04"
   OR "MAN_Q_PilotValve_05" OR "MAN_Q_PilotValve_06"
   OR "MAN_Q_PilotValve_07" OR "MAN_Q_PilotValve_08"
   OR "MAN_Q_WaterInlet_01" OR "MAN_Q_WaterInlet_02"
   OR "MAN_Q_WaterDrain";
   #AnyAutoOutput := "AUTO_Q_Heater1" OR "AUTO_Q_Heater2" OR "AUTO_Q_Heater3"
   OR "AUTO_Q_WaterPump" OR "AUTO_Q_VacuumPump"
   OR "AUTO_Q_PilotValve_01" OR "AUTO_Q_PilotValve_02"
   OR "AUTO_Q_PilotValve_03" OR "AUTO_Q_PilotValve_04"
   OR "AUTO_Q_PilotValve_05" OR "AUTO_Q_PilotValve_06"
   OR "AUTO_Q_PilotValve_07" OR "AUTO_Q_PilotValve_08"
   OR "AUTO_Q_WaterInlet_01" OR "AUTO_Q_WaterInlet_02"
   OR "AUTO_Q_WaterDrain";

   "DO_LampRun" := (#ManualMode AND #AnyManualOutput)
   OR (#AutoMode AND ("HMI_Sts_CycleRunning" OR #AnyAutoOutput));

   "DO_LampError" :="HMI_Sts_LampErrorRequest"
   OR ("HMI_Mode_Manual" AND "HMI_Mode_Auto")
   OR NOT "DI_EStop_Chain_OK"
   OR NOT "DI_Phase_OK";

   "DO_LampDoor1" := "DI_Door1_Closed";
   "DO_LampDoor2" := "DI_Door2_Closed";
END_FUNCTION

FUNCTION "FC_ProgramSelect" : Void   // FC2, SCL
{ S7_Optimized_Access := 'TRUE' }
VERSION : 0.4
   VAR_INPUT
      P1_Temp_C : Int;
      P1_Sterilize_min : Int;
      P1_DryEnable : Bool;
      P1_Dry_min : Int;
      P2_Temp_C : Int;
      P2_Sterilize_min : Int;
      P2_DryEnable : Bool;
      P2_Dry_min : Int;
      P3_Temp_C : Int;
      P3_Sterilize_min : Int;
      P3_DryEnable : Bool;
      P3_Dry_min : Int;
      P4_Temp_C : Int;
      P4_Sterilize_min : Int;
      P4_DryEnable : Bool;
      P4_Dry_min : Int;
      P5_Temp_C : Int;
      P5_Sterilize_min : Int;
      P5_DryEnable : Bool;
      P5_Dry_min : Int;   // HMI writes 1..5=recipe, 6=User, 7=Confirm User, 8=Cancel. The FC clears this command to zero after handling it.
   END_VAR
   VAR_IN_OUT
      HMI_Command : Int;
      HMI_UserTemp_C : Int;
      HMI_UserSterilize_min : Int;
      HMI_UserDryEnable : Bool;
      HMI_UserDry_min : Int;   // Persistent PLC tags / DB fields. Read these in the cycle block.
      SP_Temp_C : Real;
      SP_Sterilize_min : Int;
      SP_DryEnable : Bool;
      SP_Dry_min : Int;
      HMI_SelectedProgram : Int;
   END_VAR
   VAR_TEMP
      Temp_C : Int;
      Sterilize_min : Int;
      DryEnable : Bool;
      Dry_min : Int;
   END_VAR
BEGIN
       // Write clamped values back into the same HMI tags. Input fields
       // will show the corrected value after the PLC/HMI refresh.
       IF #HMI_UserTemp_C < 110 THEN
           #HMI_UserTemp_C := 110;
       ELSIF #HMI_UserTemp_C > 134 THEN
           #HMI_UserTemp_C := 134;
       END_IF;

       IF #HMI_UserSterilize_min < 1 THEN
           #HMI_UserSterilize_min := 1;
       ELSIF #HMI_UserSterilize_min > 99 THEN
           #HMI_UserSterilize_min := 99;
       END_IF;

       IF #HMI_UserDry_min < 0 THEN
           #HMI_UserDry_min := 0;
       ELSIF #HMI_UserDry_min > 99 THEN
           #HMI_UserDry_min := 99;
       END_IF;

       IF (#HMI_Command >= 1) AND (#HMI_Command <= 5) THEN
           CASE #HMI_Command OF
               1:
                   #Temp_C := #P1_Temp_C;
                   #Sterilize_min := #P1_Sterilize_min;
                   #DryEnable := #P1_DryEnable;
                   #Dry_min := #P1_Dry_min;
               2:
                   #Temp_C := #P2_Temp_C;
                   #Sterilize_min := #P2_Sterilize_min;
                   #DryEnable := #P2_DryEnable;
                   #Dry_min := #P2_Dry_min;
               3:
                   #Temp_C := #P3_Temp_C;
                   #Sterilize_min := #P3_Sterilize_min;
                   #DryEnable := #P3_DryEnable;
                   #Dry_min := #P3_Dry_min;
               4:
                   #Temp_C := #P4_Temp_C;
                   #Sterilize_min := #P4_Sterilize_min;
                   #DryEnable := #P4_DryEnable;
                   #Dry_min := #P4_Dry_min;
               5:
                   #Temp_C := #P5_Temp_C;
                   #Sterilize_min := #P5_Sterilize_min;
                   #DryEnable := #P5_DryEnable;
                   #Dry_min := #P5_Dry_min;
           END_CASE;

           IF (#Temp_C >= 110) AND (#Temp_C <= 134)
               AND (#Sterilize_min >= 1) AND (#Sterilize_min <= 99)
               AND (#Dry_min >= 0) AND (#Dry_min <= 99) THEN
               #SP_Temp_C := INT_TO_REAL(#Temp_C);
               #SP_Sterilize_min := #Sterilize_min;
               #SP_DryEnable := #DryEnable;
               IF #SP_DryEnable THEN
                   #SP_Dry_min := #Dry_min;
               ELSE
                   #SP_Dry_min := 0;
               END_IF;
           ELSE
               #SP_Temp_C := 0.0;
               #SP_Sterilize_min := 0;
               #SP_DryEnable := FALSE;
               #SP_Dry_min := 0;
           END_IF;

       ELSIF #HMI_Command = 6 THEN
           #SP_Temp_C := 0;
           #SP_Sterilize_min := 0;
           #SP_DryEnable := FALSE;
           #SP_Dry_min := 0;

       ELSIF #HMI_Command = 7 THEN
           #SP_Temp_C := INT_TO_REAL(#HMI_UserTemp_C);
           #SP_Sterilize_min := #HMI_UserSterilize_min;
           #SP_DryEnable := #HMI_UserDryEnable;

           IF #SP_DryEnable THEN
               #SP_Dry_min := #HMI_UserDry_min;
           ELSE
               #SP_Dry_min := 0;
           END_IF;

       ELSIF #HMI_Command = 8 THEN
           #SP_Temp_C := 0.0;
           #SP_Sterilize_min := 0;
           #SP_DryEnable := FALSE;
           #SP_Dry_min := 0;
       END_IF;

       IF #HMI_Command <> 0 THEN
           #HMI_SelectedProgram := #HMI_Command;
           #HMI_Command := 0;
       END_IF;
END_FUNCTION

ORGANIZATION_BLOCK "Main"   // OB1, LAD, ProgramCycle
TITLE = "Main Program Sweep (Cycle)"
{ S7_Optimized_Access := 'TRUE' }
VERSION : 0.1
   VAR_INPUT
      Initial_Call : Bool;   // Initial call of this OB
      Remanence : Bool;   // =True, if remanent data are available
   END_VAR
BEGIN

REGION Network 1: Analog scale
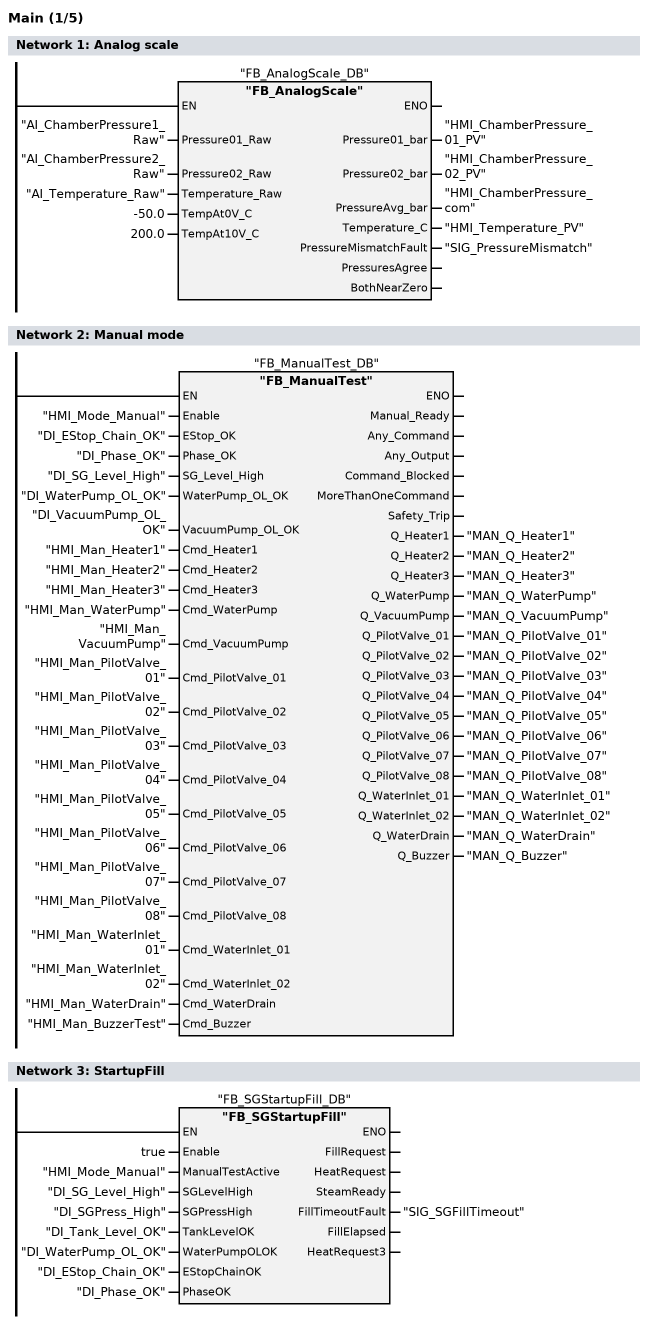
   RUNG wire#powerrail
      "FB_AnalogScale_DB"(Pressure01_Raw := "AI_ChamberPressure1_Raw", Pressure02_Raw := "AI_ChamberPressure2_Raw", Temperature_Raw := "AI_Temperature_Raw", TempAt0V_C := -50.0, TempAt10V_C := 200.0, Pressure01_bar => "HMI_ChamberPressure_01_PV", Pressure02_bar => "HMI_ChamberPressure_02_PV", PressureAvg_bar => "HMI_ChamberPressure_com", Temperature_C => "HMI_Temperature_PV", PressureMismatchFault => "SIG_PressureMismatch", PressuresAgree =>, BothNearZero =>)
   END_RUNG
   // the same network as SCL:
   "FB_AnalogScale_DB"(Pressure01_Raw := "AI_ChamberPressure1_Raw",   // "FB_AnalogScale"
                       Pressure02_Raw := "AI_ChamberPressure2_Raw",
                       Temperature_Raw := "AI_Temperature_Raw",
                       TempAt0V_C := -50.0,
                       TempAt10V_C := 200.0,
                       Pressure01_bar => "HMI_ChamberPressure_01_PV",
                       Pressure02_bar => "HMI_ChamberPressure_02_PV",
                       PressureAvg_bar => "HMI_ChamberPressure_com",
                       Temperature_C => "HMI_Temperature_PV",
                       PressureMismatchFault => "SIG_PressureMismatch");
END_REGION

REGION Network 2: Manual mode
   RUNG wire#powerrail
      "FB_ManualTest_DB"(Enable := "HMI_Mode_Manual", EStop_OK := "DI_EStop_Chain_OK", Phase_OK := "DI_Phase_OK", SG_Level_High := "DI_SG_Level_High", WaterPump_OL_OK := "DI_WaterPump_OL_OK", VacuumPump_OL_OK := "DI_VacuumPump_OL_OK", Cmd_Heater1 := "HMI_Man_Heater1", Cmd_Heater2 := "HMI_Man_Heater2", Cmd_Heater3 := "HMI_Man_Heater3", Cmd_WaterPump := "HMI_Man_WaterPump", Cmd_VacuumPump := "HMI_Man_VacuumPump", Cmd_PilotValve_01 := "HMI_Man_PilotValve_01", Cmd_PilotValve_02 := "HMI_Man_PilotValve_02", Cmd_PilotValve_03 := "HMI_Man_PilotValve_03", Cmd_PilotValve_04 := "HMI_Man_PilotValve_04", Cmd_PilotValve_05 := "HMI_Man_PilotValve_05", Cmd_PilotValve_06 := "HMI_Man_PilotValve_06", Cmd_PilotValve_07 := "HMI_Man_PilotValve_07", Cmd_PilotValve_08 := "HMI_Man_PilotValve_08", Cmd_WaterInlet_01 := "HMI_Man_WaterInlet_01", Cmd_WaterInlet_02 := "HMI_Man_WaterInlet_02", Cmd_WaterDrain := "HMI_Man_WaterDrain", Cmd_Buzzer := "HMI_Man_BuzzerTest", Manual_Ready =>, Any_Command =>, Any_Output =>, Command_Blocked =>, MoreThanOneCommand =>, Safety_Trip =>, Q_Heater1 => "MAN_Q_Heater1", Q_Heater2 => "MAN_Q_Heater2", Q_Heater3 => "MAN_Q_Heater3", Q_WaterPump => "MAN_Q_WaterPump", Q_VacuumPump => "MAN_Q_VacuumPump", Q_PilotValve_01 => "MAN_Q_PilotValve_01", Q_PilotValve_02 => "MAN_Q_PilotValve_02", Q_PilotValve_03 => "MAN_Q_PilotValve_03", Q_PilotValve_04 => "MAN_Q_PilotValve_04", Q_PilotValve_05 => "MAN_Q_PilotValve_05", Q_PilotValve_06 => "MAN_Q_PilotValve_06", Q_PilotValve_07 => "MAN_Q_PilotValve_07", Q_PilotValve_08 => "MAN_Q_PilotValve_08", Q_WaterInlet_01 => "MAN_Q_WaterInlet_01", Q_WaterInlet_02 => "MAN_Q_WaterInlet_02", Q_WaterDrain => "MAN_Q_WaterDrain", Q_Buzzer => "MAN_Q_Buzzer")
   END_RUNG
   // the same network as SCL:
   "FB_ManualTest_DB"(Enable := "HMI_Mode_Manual",   // "FB_ManualTest"
                      EStop_OK := "DI_EStop_Chain_OK",
                      Phase_OK := "DI_Phase_OK",
                      SG_Level_High := "DI_SG_Level_High",
                      WaterPump_OL_OK := "DI_WaterPump_OL_OK",
                      VacuumPump_OL_OK := "DI_VacuumPump_OL_OK",
                      Cmd_Heater1 := "HMI_Man_Heater1",
                      Cmd_Heater2 := "HMI_Man_Heater2",
                      Cmd_Heater3 := "HMI_Man_Heater3",
                      Cmd_WaterPump := "HMI_Man_WaterPump",
                      Cmd_VacuumPump := "HMI_Man_VacuumPump",
                      Cmd_PilotValve_01 := "HMI_Man_PilotValve_01",
                      Cmd_PilotValve_02 := "HMI_Man_PilotValve_02",
                      Cmd_PilotValve_03 := "HMI_Man_PilotValve_03",
                      Cmd_PilotValve_04 := "HMI_Man_PilotValve_04",
                      Cmd_PilotValve_05 := "HMI_Man_PilotValve_05",
                      Cmd_PilotValve_06 := "HMI_Man_PilotValve_06",
                      Cmd_PilotValve_07 := "HMI_Man_PilotValve_07",
                      Cmd_PilotValve_08 := "HMI_Man_PilotValve_08",
                      Cmd_WaterInlet_01 := "HMI_Man_WaterInlet_01",
                      Cmd_WaterInlet_02 := "HMI_Man_WaterInlet_02",
                      Cmd_WaterDrain := "HMI_Man_WaterDrain",
                      Cmd_Buzzer := "HMI_Man_BuzzerTest",
                      Q_Heater1 => "MAN_Q_Heater1",
                      Q_Heater2 => "MAN_Q_Heater2",
                      Q_Heater3 => "MAN_Q_Heater3",
                      Q_WaterPump => "MAN_Q_WaterPump",
                      Q_VacuumPump => "MAN_Q_VacuumPump",
                      Q_PilotValve_01 => "MAN_Q_PilotValve_01",
                      Q_PilotValve_02 => "MAN_Q_PilotValve_02",
                      Q_PilotValve_03 => "MAN_Q_PilotValve_03",
                      Q_PilotValve_04 => "MAN_Q_PilotValve_04",
                      Q_PilotValve_05 => "MAN_Q_PilotValve_05",
                      Q_PilotValve_06 => "MAN_Q_PilotValve_06",
                      Q_PilotValve_07 => "MAN_Q_PilotValve_07",
                      Q_PilotValve_08 => "MAN_Q_PilotValve_08",
                      Q_WaterInlet_01 => "MAN_Q_WaterInlet_01",
                      Q_WaterInlet_02 => "MAN_Q_WaterInlet_02",
                      Q_WaterDrain => "MAN_Q_WaterDrain",
                      Q_Buzzer => "MAN_Q_Buzzer");
END_REGION

REGION Network 3: StartupFill
   RUNG wire#powerrail
      "FB_SGStartupFill_DB"(Enable := true, ManualTestActive := "HMI_Mode_Manual", SGLevelHigh := "DI_SG_Level_High", SGPressHigh := "DI_SGPress_High", TankLevelOK := "DI_Tank_Level_OK", WaterPumpOLOK := "DI_WaterPump_OL_OK", EStopChainOK := "DI_EStop_Chain_OK", PhaseOK := "DI_Phase_OK", FillRequest =>, HeatRequest =>, SteamReady =>, FillTimeoutFault => "SIG_SGFillTimeout", FillElapsed =>, HeatRequest3 =>)
   END_RUNG
   // the same network as SCL:
   "FB_SGStartupFill_DB"(Enable := true,   // "FB_SGStartupFill"
                         ManualTestActive := "HMI_Mode_Manual",
                         SGLevelHigh := "DI_SG_Level_High",
                         SGPressHigh := "DI_SGPress_High",
                         TankLevelOK := "DI_Tank_Level_OK",
                         WaterPumpOLOK := "DI_WaterPump_OL_OK",
                         EStopChainOK := "DI_EStop_Chain_OK",
                         PhaseOK := "DI_Phase_OK",
                         FillTimeoutFault => "SIG_SGFillTimeout");
END_REGION

REGION Network 4: Alarm
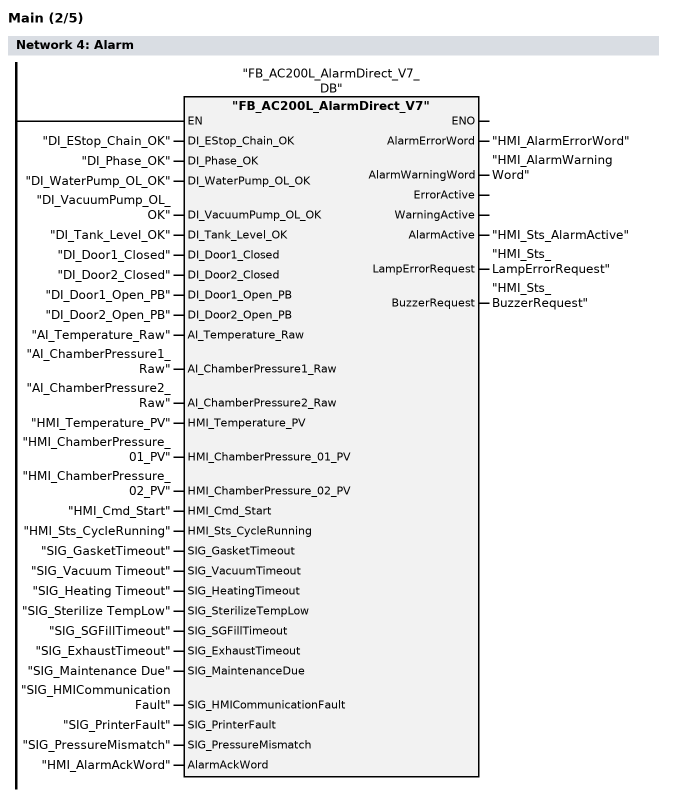
   RUNG wire#powerrail
      "FB_AC200L_AlarmDirect_V7_DB"(DI_EStop_Chain_OK := "DI_EStop_Chain_OK", DI_Phase_OK := "DI_Phase_OK", DI_WaterPump_OL_OK := "DI_WaterPump_OL_OK", DI_VacuumPump_OL_OK := "DI_VacuumPump_OL_OK", DI_Tank_Level_OK := "DI_Tank_Level_OK", DI_Door1_Closed := "DI_Door1_Closed", DI_Door2_Closed := "DI_Door2_Closed", DI_Door1_Open_PB := "DI_Door1_Open_PB", DI_Door2_Open_PB := "DI_Door2_Open_PB", AI_Temperature_Raw := "AI_Temperature_Raw", AI_ChamberPressure1_Raw := "AI_ChamberPressure1_Raw", AI_ChamberPressure2_Raw := "AI_ChamberPressure2_Raw", HMI_Temperature_PV := "HMI_Temperature_PV", HMI_ChamberPressure_01_PV := "HMI_ChamberPressure_01_PV", HMI_ChamberPressure_02_PV := "HMI_ChamberPressure_02_PV", HMI_Cmd_Start := "HMI_Cmd_Start", HMI_Sts_CycleRunning := "HMI_Sts_CycleRunning", SIG_GasketTimeout := "SIG_GasketTimeout", SIG_VacuumTimeout := "SIG_Vacuum Timeout", SIG_HeatingTimeout := "SIG_Heating Timeout", SIG_SterilizeTempLow := "SIG_Sterilize TempLow", SIG_SGFillTimeout := "SIG_SGFillTimeout", SIG_ExhaustTimeout := "SIG_ExhaustTimeout", SIG_MaintenanceDue := "SIG_Maintenance Due", SIG_HMICommunicationFault := "SIG_HMICommunicationFault", SIG_PrinterFault := "SIG_PrinterFault", SIG_PressureMismatch := "SIG_PressureMismatch", AlarmAckWord := "HMI_AlarmAckWord", AlarmErrorWord => "HMI_AlarmErrorWord", AlarmWarningWord => "HMI_AlarmWarningWord", ErrorActive =>, WarningActive =>, AlarmActive => "HMI_Sts_AlarmActive", LampErrorRequest => "HMI_Sts_LampErrorRequest", BuzzerRequest => "HMI_Sts_BuzzerRequest")
   END_RUNG
   // the same network as SCL:
   "FB_AC200L_AlarmDirect_V7_DB"(DI_EStop_Chain_OK := "DI_EStop_Chain_OK",   // "FB_AC200L_AlarmDirect_V7"
                           DI_Phase_OK := "DI_Phase_OK",
                           DI_WaterPump_OL_OK := "DI_WaterPump_OL_OK",
                           DI_VacuumPump_OL_OK := "DI_VacuumPump_OL_OK",
                           DI_Tank_Level_OK := "DI_Tank_Level_OK",
                           DI_Door1_Closed := "DI_Door1_Closed",
                           DI_Door2_Closed := "DI_Door2_Closed",
                           DI_Door1_Open_PB := "DI_Door1_Open_PB",
                           DI_Door2_Open_PB := "DI_Door2_Open_PB",
                           AI_Temperature_Raw := "AI_Temperature_Raw",
                           AI_ChamberPressure1_Raw := "AI_ChamberPressure1_Raw",
                           AI_ChamberPressure2_Raw := "AI_ChamberPressure2_Raw",
                           HMI_Temperature_PV := "HMI_Temperature_PV",
                           HMI_ChamberPressure_01_PV := "HMI_ChamberPressure_01_PV",
                           HMI_ChamberPressure_02_PV := "HMI_ChamberPressure_02_PV",
                           HMI_Cmd_Start := "HMI_Cmd_Start",
                           HMI_Sts_CycleRunning := "HMI_Sts_CycleRunning",
                           SIG_GasketTimeout := "SIG_GasketTimeout",
                           SIG_VacuumTimeout := "SIG_Vacuum Timeout",
                           SIG_HeatingTimeout := "SIG_Heating Timeout",
                           SIG_SterilizeTempLow := "SIG_Sterilize TempLow",
                           SIG_SGFillTimeout := "SIG_SGFillTimeout",
                           SIG_ExhaustTimeout := "SIG_ExhaustTimeout",
                           SIG_MaintenanceDue := "SIG_Maintenance Due",
                           SIG_HMICommunicationFault := "SIG_HMICommunicationFault",
                           SIG_PrinterFault := "SIG_PrinterFault",
                           SIG_PressureMismatch := "SIG_PressureMismatch",
                           AlarmAckWord := "HMI_AlarmAckWord",
                           AlarmErrorWord => "HMI_AlarmErrorWord",
                           AlarmWarningWord => "HMI_AlarmWarningWord",
                           AlarmActive => "HMI_Sts_AlarmActive",
                           LampErrorRequest => "HMI_Sts_LampErrorRequest",
                           BuzzerRequest => "HMI_Sts_BuzzerRequest");
END_REGION

REGION Network 5: Program Select
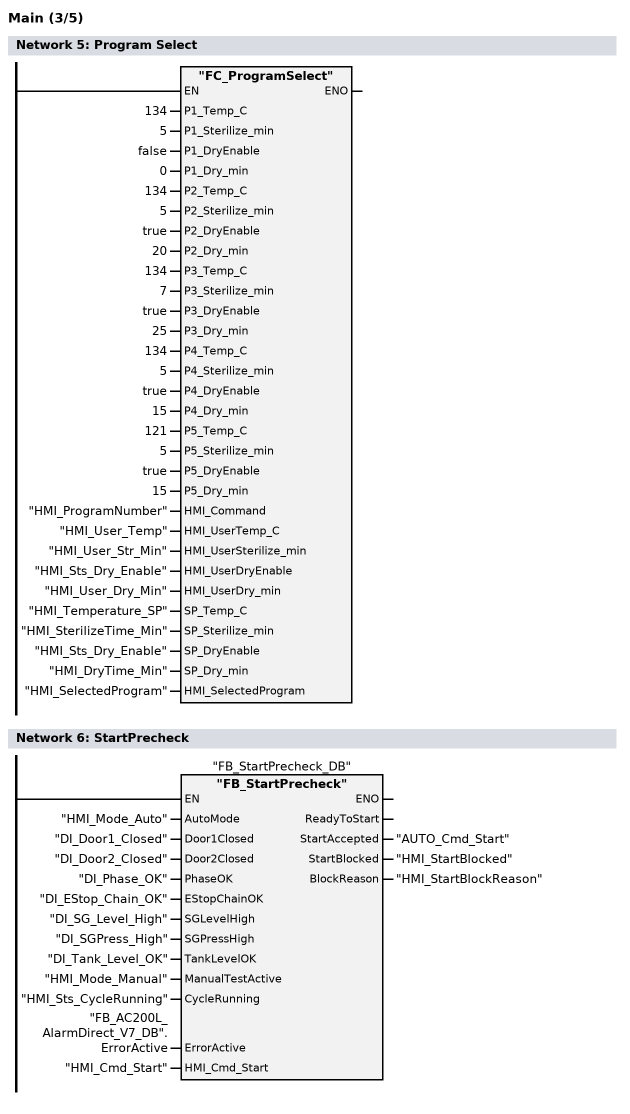
   RUNG wire#powerrail
      "FC_ProgramSelect"(P1_Temp_C := 134, P1_Sterilize_min := 5, P1_DryEnable := false, P1_Dry_min := 0, P2_Temp_C := 134, P2_Sterilize_min := 5, P2_DryEnable := true, P2_Dry_min := 20, P3_Temp_C := 134, P3_Sterilize_min := 7, P3_DryEnable := true, P3_Dry_min := 25, P4_Temp_C := 134, P4_Sterilize_min := 5, P4_DryEnable := true, P4_Dry_min := 15, P5_Temp_C := 121, P5_Sterilize_min := 5, P5_DryEnable := true, P5_Dry_min := 15, HMI_Command := "HMI_ProgramNumber", HMI_UserTemp_C := "HMI_User_Temp", HMI_UserSterilize_min := "HMI_User_Str_Min", HMI_UserDryEnable := "HMI_Sts_Dry_Enable", HMI_UserDry_min := "HMI_User_Dry_Min", SP_Temp_C := "HMI_Temperature_SP", SP_Sterilize_min := "HMI_SterilizeTime_Min", SP_DryEnable := "HMI_Sts_Dry_Enable", SP_Dry_min := "HMI_DryTime_Min", HMI_SelectedProgram := "HMI_SelectedProgram")
   END_RUNG
   // the same network as SCL:
   "FC_ProgramSelect"(P1_Temp_C := 134,
                      P1_Sterilize_min := 5,
                      P1_DryEnable := false,
                      P1_Dry_min := 0,
                      P2_Temp_C := 134,
                      P2_Sterilize_min := 5,
                      P2_DryEnable := true,
                      P2_Dry_min := 20,
                      P3_Temp_C := 134,
                      P3_Sterilize_min := 7,
                      P3_DryEnable := true,
                      P3_Dry_min := 25,
                      P4_Temp_C := 134,
                      P4_Sterilize_min := 5,
                      P4_DryEnable := true,
                      P4_Dry_min := 15,
                      P5_Temp_C := 121,
                      P5_Sterilize_min := 5,
                      P5_DryEnable := true,
                      P5_Dry_min := 15,
                      HMI_Command := "HMI_ProgramNumber",
                      HMI_UserTemp_C := "HMI_User_Temp",
                      HMI_UserSterilize_min := "HMI_User_Str_Min",
                      HMI_UserDryEnable := "HMI_Sts_Dry_Enable",
                      HMI_UserDry_min := "HMI_User_Dry_Min",
                      SP_Temp_C := "HMI_Temperature_SP",
                      SP_Sterilize_min := "HMI_SterilizeTime_Min",
                      SP_DryEnable := "HMI_Sts_Dry_Enable",
                      SP_Dry_min := "HMI_DryTime_Min",
                      HMI_SelectedProgram := "HMI_SelectedProgram");
END_REGION

REGION Network 6: StartPrecheck
   RUNG wire#powerrail
      "FB_StartPrecheck_DB"(AutoMode := "HMI_Mode_Auto", Door1Closed := "DI_Door1_Closed", Door2Closed := "DI_Door2_Closed", PhaseOK := "DI_Phase_OK", EStopChainOK := "DI_EStop_Chain_OK", SGLevelHigh := "DI_SG_Level_High", SGPressHigh := "DI_SGPress_High", TankLevelOK := "DI_Tank_Level_OK", ManualTestActive := "HMI_Mode_Manual", CycleRunning := "HMI_Sts_CycleRunning", ErrorActive := "FB_AC200L_AlarmDirect_V7_DB".ErrorActive, HMI_Cmd_Start := "HMI_Cmd_Start", ReadyToStart =>, StartAccepted => "AUTO_Cmd_Start", StartBlocked => "HMI_StartBlocked", BlockReason => "HMI_StartBlockReason")
   END_RUNG
   // the same network as SCL:
   "FB_StartPrecheck_DB"(AutoMode := "HMI_Mode_Auto",   // "FB_StartPrecheck"
                         Door1Closed := "DI_Door1_Closed",
                         Door2Closed := "DI_Door2_Closed",
                         PhaseOK := "DI_Phase_OK",
                         EStopChainOK := "DI_EStop_Chain_OK",
                         SGLevelHigh := "DI_SG_Level_High",
                         SGPressHigh := "DI_SGPress_High",
                         TankLevelOK := "DI_Tank_Level_OK",
                         ManualTestActive := "HMI_Mode_Manual",
                         CycleRunning := "HMI_Sts_CycleRunning",
                         ErrorActive := "FB_AC200L_AlarmDirect_V7_DB".ErrorActive,
                         HMI_Cmd_Start := "HMI_Cmd_Start",
                         StartAccepted => "AUTO_Cmd_Start",
                         StartBlocked => "HMI_StartBlocked",
                         BlockReason => "HMI_StartBlockReason");
END_REGION

